	{attribute 'export' := '("archive":"True","name":"АОсс: АОсс от оператора","alarm":("type":"crs","action":"АОсс"),"subsystem":"Внешние источники","condition":("set":"TRUE","reset":"FALSE","active":"btn.AOss.out","fault":"FALSE"))'}
	btn_AOss : Tcrs:= (subsystem_num := 1, type_num := 1); //АОсс: АОсс от оператора//ALG/Внешние источники
	{attribute 'export' := '("archive":"True","name":"АОбс: АОбс от оператора","alarm":("type":"crs","action":"АОбс"),"subsystem":"Внешние источники","condition":("set":"TRUE","reset":"FALSE","active":"btn.AObs.out","fault":"FALSE"))'}
	btn_AObs : Tcrs:= (subsystem_num := 1, type_num := 2); //АОбс: АОбс от оператора//ALG/Внешние источники
	{attribute 'export' := '("archive":"True","name":"АОсс: АОсс по технологическим условиям","alarm":("type":"crs","action":"АОсс"),"subsystem":"Внешние источники","condition":("set":"TRUE","reset":"FALSE","active":"alg.AOss_tech","fault":"FALSE"))'}
	AOss_tech : Tcrs:= (subsystem_num := 1, type_num := 1); //АОсс: АОсс по технологическим условиям//ALG/Внешние источники
	{attribute 'export' := '("archive":"True","name":"АОбс: АОбс по технологическим условиям","alarm":("type":"crs","action":"АОбс"),"subsystem":"Внешние источники","condition":("set":"TRUE","reset":"FALSE","active":"alg.AOss_tech","fault":"FALSE"))'}
	AObs_tech : Tcrs:= (subsystem_num := 1, type_num := 2); //АОбс: АОбс по технологическим условиям//ALG/Внешние источники
	{attribute 'export' := '("archive":"True","name":"АОсс: Кнопка АО на ПРУ","alarm":("type":"crs","action":"АОсс"),"subsystem":"Внешние источники","condition":("set":"TRUE","reset":"FALSE","active":"dipar.AO_PRU_1.value OR dipar.AO_PRU_2.value","fault":"dipar.AO_PRU_1.flt OR dipar.AO_PRU_2.flt"))'}
	AO_PRU : Tcrs:= (subsystem_num := 1, type_num := 1); //АОсс: Кнопка АО на ПРУ//ALG/Внешние источники
	{attribute 'export' := '("archive":"True","name":"АОсс: АО от кнопки \"АО\" блока автоматики ГПА","alarm":("type":"crs","action":"АОсс"),"subsystem":"Внешние источники","condition":("set":"TRUE","reset":"FALSE","active":"dipar.AO_BA.value","fault":"dipar.AO_BA.flt"))'}
	AO_BA : Tcrs:= (subsystem_num := 1, type_num := 1); //АОсс: АО от кнопки "АО" блока автоматики ГПА//DI/Внешние источники
	{attribute 'export' := '("archive":"True","name":"АОсс: БЭАО сработал","alarm":("type":"crs","action":"АОсс"),"subsystem":"Внешние источники","condition":("set":"TRUE","reset":"FALSE","active":"dipar.BEAO.value","fault":"dipar.BEAO.flt"))'}
	BEAO : Tcrs:= (subsystem_num := 1, type_num := 1); //АОсс: БЭАО сработал//DI/Внешние источники
	{attribute 'export' := '("archive":"True","name":"АОбс: Самопроизвольное закрытие СК","alarm":("type":"crs","action":"АОбс"),"subsystem":"Блок двигателя","condition":("set":"FuelReg.fReg.isFire","reset":"NOT am.SK.on","active":"NOT dipar.SK_ON.value","fault":"dipar.SK_ON.flt"))'}
	Causeless_SK : Tcrs:= (subsystem_num := 2, type_num := 2); //АОбс: Самопроизвольное закрытие СК//ALG/Блок двигателя
	{attribute 'export' := '("archive":"True","name":"АОсс: Помпаж двигателя","alarm":("type":"crs","action":"АОсс"),"subsystem":"Блок двигателя","condition":("set":"TRUE","reset":"FALSE","active":"dipar.SurgeD.value","fault":"dipar.SurgeD.flt"))'}
	SurgeD : Tcrs:= (subsystem_num := 2, type_num := 1); //АОсс: Помпаж двигателя//DI/Блок двигателя
	{attribute 'export' := '("archive":"True","name":"АОсс: Опасная вибрация двигателя","alarm":("type":"crs","action":"АОсс"),"subsystem":"Блок двигателя","condition":("set":"TRUE","reset":"FALSE","active":"dipar.Vs_D_Av.value","fault":"dipar.Vs_D_Av.flt"))'}
	Vs_D_Av : Tcrs:= (subsystem_num := 2, type_num := 1); //АОсс: Опасная вибрация двигателя//DI/Блок двигателя
	{attribute 'export' := '("archive":"True","name":"АОбс: Авар.-выс. Вибрация ТК","alarm":("type":"crs","action":"АОбс"),"subsystem":"Блок двигателя","condition":("set":"TRUE","reset":"FALSE","active":"aipar.Vstk.setpoint.HH","fault":"aipar.Vstk.flt"))'}
	Vstk_HH : Tcrs:= (subsystem_num := 2, type_num := 2); //АОбс: Авар.-выс. Вибрация ТК//> 60/Блок двигателя
	{attribute 'export' := '("archive":"True","name":"АОсс: Авар.-выс. Вибрация СТ","alarm":("type":"crs","action":"АОсс"),"subsystem":"Блок двигателя","condition":("set":"TRUE","reset":"FALSE","active":"aipar.Vsst.setpoint.HH","fault":"aipar.Vsst.flt"))'}
	Vsst_HH : Tcrs:= (subsystem_num := 2, type_num := 1); //АОсс: Авар.-выс. Вибрация СТ//> 60/Блок двигателя
	{attribute 'export' := '("archive":"True","name":"АОбс: КПВ234 не закрыты","alarm":("type":"crs","action":"АОбс"),"subsystem":"Блок двигателя","condition":("set":"alg.KPV234_wOpen","reset":"NOT alg.KPV234_wOpen","active":"NOT ( dipar.KPV2_off.value AND dipar.KPV3_off.value AND dipar.KPV4_off.value )","fault":"dipar.KPV2_off.flt OR dipar.KPV3_off.flt OR dipar.KPV4_off.flt"))'}
	KPV234_wOpen : Tcrs:= (subsystem_num := 2, type_num := 2, pt := t#1s0ms); //АОбс: КПВ234 не закрыты//ALG/Блок двигателя
	{attribute 'export' := '("archive":"True","name":"АОбс: КПВ15 не закрыты","alarm":("type":"crs","action":"АОбс"),"subsystem":"Блок двигателя","condition":("set":"alg.KPV15_wOpen","reset":"NOT alg.KPV15_wOpen","active":"NOT ( dipar.KPV1_off.value AND dipar.KPV5_off.value )","fault":"dipar.KPV1_off.flt OR dipar.KPV5_off.flt"))'}
	KPV15_wOpen : Tcrs:= (subsystem_num := 2, type_num := 2, pt := t#1s0ms); //АОбс: КПВ15 не закрыты//ALG/Блок двигателя
	{attribute 'export' := '("archive":"True","name":"АОбс: КПВ15 не открыты","alarm":("type":"crs","action":"АОбс"),"subsystem":"Блок двигателя","condition":("set":"alg.KPV15_nOpen","reset":"NOT alg.KPV15_nOpen","active":"NOT ( dipar.KPV1_ON.value AND dipar.KPV5_ON.value )","fault":"dipar.KPV1_ON.flt OR dipar.KPV5_ON.flt"))'}
	KPV15_nOpen : Tcrs:= (subsystem_num := 2, type_num := 2, pt := t#1s0ms); //АОбс: КПВ15 не открыты//ALG/Блок двигателя
	{attribute 'export' := '("archive":"True","name":"АОсс: Авар.-выс. Обороты СТ > 9300 об/мин","alarm":("type":"crs","action":"АОсс"),"subsystem":"Блок двигателя","condition":("set":"TRUE","reset":"FALSE","active":"acpar.Nst.setpoint.HH","fault":"FALSE"))'}
	Nst_HH : Tcrs:= (subsystem_num := 2, type_num := 1); //АОсс: Авар.-выс. Обороты СТ > 9300 об/мин//> 9000 об/мин/Блок двигателя
	{attribute 'export' := '("archive":"True","name":"АОбс: Авар.-выс. Обороты ТК > 8400 об/мин","alarm":("type":"crs","action":"АОбс"),"subsystem":"Блок двигателя","condition":("set":"TRUE","reset":"FALSE","active":"acpar.Ntk.setpoint.HH","fault":"FALSE"))'}
	Ntk_Av_HH : Tcrs:= (subsystem_num := 2, type_num := 2); //АОбс: Авар.-выс. Обороты ТК > 8400 об/мин//> 8400 об/мин/Блок двигателя
	{attribute 'export' := '("archive":"True","name":"АОбс: Отказ всех датчиков ЧВ ТК","alarm":("type":"crs","action":"АОбс"),"subsystem":"Блок двигателя","condition":("set":"TRUE","reset":"FALSE","active":"aipar.Ntk_1.flt AND aipar.Ntk_2.flt OR acpar.Ntk.flt","fault":"FALSE"))'}
	Ntk_flt : Tcrs:= (subsystem_num := 2, type_num := 2); //АОбс: Отказ всех датчиков ЧВ ТК//ALG/Блок двигателя
	{attribute 'export' := '("archive":"True","name":"АОбс: Отказ всех датчиков ЧВ СТ","alarm":("type":"crs","action":"АОбс"),"subsystem":"Блок двигателя","condition":("set":"TRUE","reset":"FALSE","active":"aipar.Nst_1.flt AND aipar.Nst_2.flt OR acpar.Nst.flt","fault":"FALSE"))'}
	Nst_flt : Tcrs:= (subsystem_num := 2, type_num := 2); //АОбс: Отказ всех датчиков ЧВ СТ//ALG/Блок двигателя
	{attribute 'export' := '("archive":"True","name":"АОбс: Авар.-выс. Температура газа на входе СТ","alarm":("type":"crs","action":"АОбс"),"subsystem":"Блок двигателя","condition":("set":"TRUE","reset":"FALSE","active":"acpar.Tg_inST.setpoint.HH","fault":"FALSE"))'}
	Tg_inST_HH : Tcrs:= (subsystem_num := 2, type_num := 2); //АОбс: Авар.-выс. Температура газа на входе СТ//> 670 °С/Блок двигателя
	{attribute 'export' := '("archive":"True","name":"АОсс: Пожар ОД","alarm":("type":"crs","action":"АОсс"),"subsystem":"Блок двигателя","condition":("set":"TRUE","reset":"FALSE","active":"dipar.Fire_OD.value","fault":"dipar.Fire_OD.flt"))'}
	Fire_OD : Tcrs:= (subsystem_num := 2, type_num := 1); //АОсс: Пожар ОД//DI/Блок двигателя
	{attribute 'export' := '("archive":"True","name":"АОбс: Авар.-выс. Высокая неравномерность 1-ой термопары","alarm":("type":"crs","action":"АОбс"),"subsystem":"Блок двигателя","condition":("set":"am.SK.isON","reset":"am.SK.isOFF","active":"ABS ( acpar.Tg_inST.value - aipar.Tg_inST_1.value ) > 100.0","fault":"aipar.Tg_inST_1.flt"))'}
	Tg1_inSTdistort_HH : Tcrs:= (subsystem_num := 2, type_num := 2); //АОбс: Авар.-выс. Высокая неравномерность 1-ой термопары//<> 100 °С/Блок двигателя
	{attribute 'export' := '("archive":"True","name":"АОбс: Авар.-выс. Высокая неравномерность 2-ой термопары","alarm":("type":"crs","action":"АОбс"),"subsystem":"Блок двигателя","condition":("set":"am.SK.isON","reset":"am.SK.isOFF","active":"ABS ( acpar.Tg_inST.value - aipar.Tg_inST_2.value ) > 100.0","fault":"aipar.Tg_inST_2.flt"))'}
	Tg2_inSTdistort_HH : Tcrs:= (subsystem_num := 2, type_num := 2); //АОбс: Авар.-выс. Высокая неравномерность 2-ой термопары//<> 100 °С/Блок двигателя
	{attribute 'export' := '("archive":"True","name":"АОбс: Авар.-выс. Высокая неравномерность 3-ой термопары","alarm":("type":"crs","action":"АОбс"),"subsystem":"Блок двигателя","condition":("set":"am.SK.isON","reset":"am.SK.isOFF","active":"ABS ( acpar.Tg_inST.value - aipar.Tg_inST_3.value ) > 100.0","fault":"aipar.Tg_inST_3.flt"))'}
	Tg3_inSTdistort_HH : Tcrs:= (subsystem_num := 2, type_num := 2); //АОбс: Авар.-выс. Высокая неравномерность 3-ой термопары//<> 100 °С/Блок двигателя
	{attribute 'export' := '("archive":"True","name":"АОбс: Авар.-выс. Высокая неравномерность 4-ой термопары","alarm":("type":"crs","action":"АОбс"),"subsystem":"Блок двигателя","condition":("set":"am.SK.isON","reset":"am.SK.isOFF","active":"ABS ( acpar.Tg_inST.value - aipar.Tg_inST_4.value ) > 100.0","fault":"aipar.Tg_inST_4.flt"))'}
	Tg4_inSTdistort_HH : Tcrs:= (subsystem_num := 2, type_num := 2); //АОбс: Авар.-выс. Высокая неравномерность 4-ой термопары//<> 100 °С/Блок двигателя
	{attribute 'export' := '("archive":"True","name":"АОбс: Авар.-выс. Высокая неравномерность 5-ой термопары","alarm":("type":"crs","action":"АОбс"),"subsystem":"Блок двигателя","condition":("set":"am.SK.isON","reset":"am.SK.isOFF","active":"ABS ( acpar.Tg_inST.value - aipar.Tg_inST_5.value ) > 100.0","fault":"aipar.Tg_inST_5.flt"))'}
	Tg5_inSTdistort_HH : Tcrs:= (subsystem_num := 2, type_num := 2); //АОбс: Авар.-выс. Высокая неравномерность 5-ой термопары//<> 100 °С/Блок двигателя
	{attribute 'export' := '("archive":"True","name":"АОбс: Авар.-выс. Высокая неравномерность 6-ой термопары","alarm":("type":"crs","action":"АОбс"),"subsystem":"Блок двигателя","condition":("set":"am.SK.isON","reset":"am.SK.isOFF","active":"ABS ( acpar.Tg_inST.value - aipar.Tg_inST_6.value ) > 100.0","fault":"aipar.Tg_inST_6.flt"))'}
	Tg6_inSTdistort_HH : Tcrs:= (subsystem_num := 2, type_num := 2); //АОбс: Авар.-выс. Высокая неравномерность 6-ой термопары//<> 100 °С/Блок двигателя
	{attribute 'export' := '("archive":"True","name":"АОбс: Отказ 4-х и более термопар","alarm":("type":"crs","action":"АОбс"),"subsystem":"Блок двигателя","condition":("set":"TRUE","reset":"FALSE","active":"alg.TstInWork < 3","fault":"FALSE"))'}
	Tg_inSTflt : Tcrs:= (subsystem_num := 2, type_num := 2); //АОбс: Отказ 4-х и более термопар//ALG/Блок двигателя
	{attribute 'export' := '("archive":"True","name":"АОбс: Нет розжига на пуске","alarm":("type":"crs","action":"АОбс"),"subsystem":"Блок двигателя","condition":("set":"alg.sh_nIgnition","reset":"NOT alg.sh_nIgnition","active":"NOT FuelReg.fReg.isFire","fault":"FALSE"))'}
	nIgnition : Tcrs:= (subsystem_num := 2, type_num := 2, pt := t#10s0ms); //АОбс: Нет розжига на пуске//DI/Блок двигателя
	{attribute 'export' := '("archive":"True","name":"АОбс: Погасание факела","alarm":("type":"crs","action":"АОбс"),"subsystem":"Блок двигателя","condition":("set":"TRUE","reset":"FALSE","active":"FuelReg.fReg.noFire","fault":"FALSE"))'}
	Fire_flt : Tcrs:= (subsystem_num := 2, type_num := 2); //АОбс: Погасание факела//ALG/Блок двигателя
	{attribute 'export' := '("archive":"True","name":"АОбс: Отсутствие раскрутки ТК","alarm":("type":"crs","action":"АОбс"),"subsystem":"Блок двигателя","condition":("set":"alg.sh_nBoost","reset":"NOT alg.sh_nBoost","active":"acpar.Ntk.value < 5600","fault":"acpar.Ntk.flt"))'}
	Ntk_nBoost : Tcrs:= (subsystem_num := 2, type_num := 2, pt := t#10s0ms); //АОбс: Отсутствие раскрутки ТК//DI/Блок двигателя
	{attribute 'export' := '("archive":"True","name":"АОбс: Рассогласование ДГ","alarm":("type":"crs","action":"АОбс"),"subsystem":"Блок двигателя","condition":("set":"am.SK.on","reset":"NOT am.SK.on","active":"ABS(aopar.DG_set.value - aipar.DG_Pos.value) >= 1.0","fault":"aipar.DG_Pos.flt"))'}
	DGdistort : Tcrs:= (subsystem_num := 2, type_num := 2, pt := t#2s0ms); //АОбс: Рассогласование ДГ//ALG/Блок двигателя
	{attribute 'export' := '("archive":"True","name":"АОбс: Авар.-выс. Давление воздуха за 14-й ступенью осевого компрессора","alarm":("type":"crs","action":"АОбс"),"subsystem":"Блок двигателя","condition":("set":"TRUE","reset":"FALSE","active":"aipar.Pa_out14.setpoint.HH","fault":"aipar.Pa_out14.flt"))'}
	Pa_out14_HH : Tcrs:= (subsystem_num := 2, type_num := 2); //АОбс: Авар.-выс. Давление воздуха за 14-й ступенью осевого компрессора//> 2.0/Блок двигателя
	{attribute 'export' := '("archive":"True","name":"АОбс: Неисправность БЗА на пуске","alarm":("type":"crs","action":"АОбс"),"subsystem":"Блок двигателя","condition":("set":"( acpar.Ntk.value > BZA.Ntk_SetUp ) AND ( acpar.Nst.value > BZA.Nst_SetUp )","reset":"NOT tch.GTDstart.value","active":"NOT dipar.BZA_ready_1.value OR NOT dipar.BZA_ready_2.value","fault":"FALSE"))'}
	BZA_ready_2 : Tcrs:= (subsystem_num := 2, type_num := 2); //АОбс: Неисправность БЗА на пуске//DI/Блок двигателя
	{attribute 'export' := '("archive":"True","name":"АОсс: БЗА: Авария","alarm":("type":"crs","action":"АОсс"),"subsystem":"Блок двигателя","condition":("set":"TRUE","reset":"FALSE","active":"dipar.BZA_alr.value","fault":"dipar.BZA_alr.flt"))'}
	BZA_alr : Tcrs:= (subsystem_num := 2, type_num := 1); //АОсс: БЗА: Авария//DI/Блок двигателя
	{attribute 'export' := '("archive":"True","name":"АОбс: Давление масла смазки ТК аварийное","alarm":("type":"crs","action":"АОбс"),"subsystem":"Маслосистема двигателя","condition":("set":"alg.sh_PmGTD","reset":"NOT alg.sh_PmGTD","active":"dipar.Pm_TK_An.value","fault":"dipar.Pm_TK_An.flt"))'}
	Pm_TK_An : Tcrs:= (subsystem_num := 3, type_num := 2, pt := t#3s0ms); //АОбс: Давление масла смазки ТК аварийное//DI/Маслосистема двигателя
	{attribute 'export' := '("archive":"True","name":"АОбс: Давление масла смазки СТ аварийное","alarm":("type":"crs","action":"АОбс"),"subsystem":"Маслосистема двигателя","condition":("set":"alg.sh_PmGTD","reset":"NOT alg.sh_PmGTD","active":"dipar.Pm_ST_An.value","fault":"dipar.Pm_ST_An.flt"))'}
	Pm_ST_An : Tcrs:= (subsystem_num := 3, type_num := 2, pt := t#3s0ms); //АОбс: Давление масла смазки СТ аварийное//DI/Маслосистема двигателя
	{attribute 'export' := '("archive":"True","name":"АОбс: Авар.-выс. Температура масла на выходе двигателя","alarm":("type":"crs","action":"АОбс"),"subsystem":"Маслосистема двигателя","condition":("set":"TRUE","reset":"FALSE","active":"aipar.Tm_outD.setpoint.HH","fault":"aipar.Tm_outD.flt"))'}
	Tm_outD_HH : Tcrs:= (subsystem_num := 3, type_num := 2, pt := t#1s0ms); //АОбс: Авар.-выс. Температура масла на выходе двигателя//> 85 °С/Маслосистема двигателя
	{attribute 'export' := '("archive":"True","name":"АОсс: Стружка в масле на выходе Д","alarm":("type":"crs","action":"АОсс"),"subsystem":"Маслосистема двигателя","condition":("set":"TRUE","reset":"FALSE","active":"dipar.Chip_outD.value","fault":"dipar.Chip_outD.flt"))'}
	Chip_outD : Tcrs:= (subsystem_num := 3, type_num := 1); //АОсс: Стружка в масле на выходе Д//DI/Маслосистема двигателя
	{attribute 'export' := '("archive":"True","name":"АОбс: Аварийное давление газа до крана 13","alarm":("type":"crs","action":"АОбс"),"subsystem":"Воздушный стартер","condition":("set":"alg.sh_Pg_InKR13","reset":"NOT alg.sh_Pg_InKR13","active":"dipar.Pg_InKR13.value","fault":"dipar.Pg_InKR13.flt"))'}
	Pg_InKR13 : Tcrs:= (subsystem_num := 4, type_num := 2, pt := t#10s0ms); //АОбс: Аварийное давление газа до крана 13//DI/Воздушный стартер
	{attribute 'export' := '("archive":"True","name":"АОбс: Давление масла смазки воздушного стартера высокий уровень","alarm":("type":"crs","action":"АОбс"),"subsystem":"Воздушный стартер","condition":("set":"TRUE","reset":"FALSE","active":"dipar.Pm_Starter_Av.value","fault":"dipar.Pm_Starter_Av.flt"))'}
	Pm_Starter_Av : Tcrs:= (subsystem_num := 4, type_num := 2, pt := t#10s0ms); //АОбс: Давление масла смазки воздушного стартера высокий уровень//DI/Воздушный стартер
	{attribute 'export' := '("archive":"True","name":"АОбс: Давление масла смазки воздушного стартера низкий уровень","alarm":("type":"crs","action":"АОбс"),"subsystem":"Воздушный стартер","condition":("set":"alg.sh_Starter","reset":"am.KR13.isOFF","active":"dipar.Pm_Starter_An.value","fault":"dipar.Pm_Starter_An.flt"))'}
	Pm_Starter_An : Tcrs:= (subsystem_num := 4, type_num := 2); //АОбс: Давление масла смазки воздушного стартера низкий уровень//DI/Воздушный стартер
	{attribute 'export' := '("archive":"True","name":"АОбс: Давление газа перед дозатором газа Аварийное","alarm":("type":"crs","action":"АОбс"),"subsystem":"Блок топливного газа","condition":("set":"alg.sh_TG","reset":"NOT alg.sh_TG","active":"dipar.Ptg_inDG_An.value","fault":"dipar.Ptg_inDG_An.flt"))'}
	Ptg_inDG_An : Tcrs:= (subsystem_num := 6, type_num := 2, pt := t#1s0ms); //АОбс: Давление газа перед дозатором газа Аварийное//DI/Блок топливного газа
	{attribute 'export' := '("archive":"True","name":"АОсс: dP перед форсунками камеры сгорания >10кПа","alarm":("type":"crs","action":"АОсс"),"subsystem":"Блок топливного газа","condition":("set":"am.SK.isOFF AND ( acpar.Ntk.value < 100 )","reset":"am.SK.isON","active":"dipar.dP_F_Pv.value","fault":"dipar.dP_F_Pv.flt"))'}
	dP_F_Pv : Tcrs:= (subsystem_num := 6, type_num := 1, pt := t#3s0ms); //АОсс: dP перед форсунками камеры сгорания >10кПа//DI/Блок топливного газа
	{attribute 'export' := '("archive":"True","name":"АОбс: Аварийное давление масла перед ДГ","alarm":("type":"crs","action":"АОбс"),"subsystem":"Блок топливного газа","condition":("set":"alg.sh_SAR","reset":"NOT alg.sh_SAR","active":"dipar.Pm_SAR_An.value","fault":"dipar.Pm_SAR_An.flt"))'}
	Pm_SAR_An : Tcrs:= (subsystem_num := 6, type_num := 2, pt := t#1s0ms); //АОбс: Аварийное давление масла перед ДГ//DI/Блок топливного газа
	{attribute 'export' := '("archive":"True","name":"АОбс: Авар.-низ. Давление топливного газа перед ТРК","alarm":("type":"crs","action":"АОбс"),"subsystem":"Блок топливного газа","condition":("set":"alg.sh_TG","reset":"NOT alg.sh_TG","active":"aipar.Ptg_inTRK.setpoint.LL","fault":"aipar.Ptg_inTRK.flt"))'}
	Ptg_inTRK_LL : Tcrs:= (subsystem_num := 6, type_num := 2, pt := t#3s0ms); //АОбс: Авар.-низ. Давление топливного газа перед ТРК//< 10 кгс/см2/Блок топливного газа
	{attribute 'export' := '("archive":"True","name":"АОсс: Помпаж нагнетателя","alarm":("type":"crs","action":"АОсс"),"subsystem":"Компрессорная установка/блок нагнетателя","condition":("set":"TRUE","reset":"FALSE","active":"s_tunpar.ASprot.surge","fault":"s_tunpar.ASprot.surgeAlertBrk"))'}
	AS_Av : Tcrs:= (subsystem_num := 9, type_num := 1); //АОсс: Помпаж нагнетателя//DI/Компрессорная установка/блок нагнетателя
	{attribute 'export' := '("archive":"True","name":"АОсс: Авар.-низ. Перепад давления “масло-газ”","alarm":("type":"crs","action":"АОсс"),"subsystem":"Компрессорная установка/блок нагнетателя","condition":("set":"alg.sh_dPmg","reset":"NOT alg.sh_dPmg","active":"aipar.dPmg.setpoint.LL OR dipar.dPmg_An.value","fault":"dipar.dPmg_An.flt OR aipar.dPmg.flt OR NOT aipar.dPmg.setpoint.isLL"))'}
	dPmg_LL : Tcrs:= (subsystem_num := 9, type_num := 1); //АОсс: Авар.-низ. Перепад давления “масло-газ”//< 0.3 кгс/см2/Компрессорная установка/блок нагнетателя
	{attribute 'export' := '("archive":"True","name":"АОсс: Давление масла смазки Н аварийное","alarm":("type":"crs","action":"АОсс"),"subsystem":"Компрессорная установка/блок нагнетателя","condition":("set":"alg.sh_PmN","reset":"NOT alg.sh_PmN","active":"dipar.Pm_N_An.value","fault":"dipar.Pm_N_An.flt"))'}
	Pm_N_An : Tcrs:= (subsystem_num := 9, type_num := 1, pt := t#3s0ms); //АОсс: Давление масла смазки Н аварийное//DI/Компрессорная установка/блок нагнетателя
	{attribute 'export' := '("archive":"True","name":"АОсс: Аварийный осевой сдвиг ротора Н","alarm":("type":"crs","action":"АОсс"),"subsystem":"Компрессорная установка/блок нагнетателя","condition":("set":"TRUE","reset":"FALSE","active":"dipar.Zs_Nl.value","fault":"dipar.Zs_Nl.flt"))'}
	Zs_Nl : Tcrs:= (subsystem_num := 9, type_num := 1); //АОсс: Аварийный осевой сдвиг ротора Н//DI/Компрессорная установка/блок нагнетателя
	{attribute 'export' := '("archive":"True","name":"АОбс: Кран 6 закрыт на пуске","alarm":("type":"crs","action":"АОбс"),"subsystem":"Компрессорная установка/блок нагнетателя","condition":("set":"acpar.Nst.value > 300.0  AND Start_D.drm.active","reset":"acpar.Nst.value < 300.0 OR NOT Start_D.drm.active","active":"dipar.Kr6_off.value","fault":"dipar.Kr6_off.flt"))'}
	Kr6_off_start : Tcrs:= (subsystem_num := 9, type_num := 2, pt := t#3s0ms); //АОбс: Кран 6 закрыт на пуске//ALG/Компрессорная установка/блок нагнетателя
	{attribute 'export' := '("archive":"True","name":"АОбс: Самопроизвольное закрытие крана 1","alarm":("type":"crs","action":"АОбс"),"subsystem":"Газовая обвязка","condition":("set":"alg.work","reset":"NOT alg.work","active":"NOT dipar.Kr1_ON.value","fault":"FALSE"))'}
	Causeless_KR1_off : Tcrs:= (subsystem_num := 11, type_num := 2, pt := t#3s0ms); //АОбс: Самопроизвольное закрытие крана 1//ALG/Газовая обвязка
	{attribute 'export' := '("archive":"True","name":"АОбс: Самопроизвольное закрытие крана 2","alarm":("type":"crs","action":"АОбс"),"subsystem":"Газовая обвязка","condition":("set":"alg.work","reset":"NOT alg.work","active":"NOT dipar.Kr2_ON.value AND dipar.Kr6_off.value","fault":"FALSE"))'}
	Causeless_KR2_off : Tcrs:= (subsystem_num := 11, type_num := 2, pt := t#3s0ms); //АОбс: Самопроизвольное закрытие крана 2//ALG/Газовая обвязка
	{attribute 'export' := '("archive":"True","name":"АОбс: Самопроизвольное закрытие крана 6","alarm":("type":"crs","action":"АОбс"),"subsystem":"Газовая обвязка","condition":("set":"alg.work","reset":"NOT alg.work","active":"NOT dipar.Kr6_ON.value AND (NOT dipar.Kr2_ON.value OR dipar.Kr2_off.value)","fault":"FALSE"))'}
	Causeless_KR6_off : Tcrs:= (subsystem_num := 11, type_num := 2, pt := t#3s0ms); //АОбс: Самопроизвольное закрытие крана 6//ALG/Газовая обвязка
	{attribute 'export' := '("archive":"True","name":"АОбс: Самопроизвольная перестановка кранов 10, 11","alarm":("type":"crs","action":"АОбс"),"subsystem":"Газовая обвязка","condition":("set":"am.KR15.on","reset":"NOT am.KR15.on","active":"NOT ( dipar.Kr10_off.value AND dipar.Kr11_ON.value )","fault":"FALSE"))'}
	Causeless_KR10_11 : Tcrs:= (subsystem_num := 11, type_num := 2, pt := t#1s0ms); //АОбс: Самопроизвольная перестановка кранов 10, 11//ALG/Газовая обвязка
END_VAR
(* global variable list ppu *)
{region INFO}
(*
 Назначение: Признаки срабатывания предпусковых условий
 Автор:  /Andrey/ 24.06.2025 16:50:31
 Версия: v00.00.22
 Проект: KA107__GPA2
*)
{endregion}
{attribute 'qualified_only'}
{attribute 'symbol' := 'read'}
VAR_GLOBAL
	{attribute 'symbol' := 'none'}
	common: Talarm; //Общий сигнал для VAR_STAT
	{attribute 'export' := '("archive":"True","name":"Контроль ХР")'}
	check_HR: Ttch; //Контроль ХР
	{attribute 'export' := '("archive":"True","name":"Контроль ГР")'}
	check_GR: Ttch; //Контроль ГР
	{attribute 'symbol' := 'none'}
	HR: BOOL; //Условия ХР собраны
	{attribute 'symbol' := 'none'}
	GR: BOOL; //Условия ГР собраны

	{attribute 'export' := '("archive":"True","name":"Есть недеблокированные АС","alarm":("type":"ppu","action":"ХР"),"condition":("set":"TRUE","reset":"FALSE","active":"crs.common.aggregated"))'}
	crs_aggregated : Talarm:= (subsystem_num := 1, type_num := 4); //Есть недеблокированные АС//Внутренний сигнал/Внешние источники
	{attribute 'export' := '("archive":"True","name":"Расчетная N ротора ГГ > 100 об/мин","alarm":("type":"ppu","action":"ХР"),"condition":("set":"TRUE","reset":"FALSE","active":"acpar.Ntk.value > 100.0"))'}
	evNvd_H : Talarm:= (subsystem_num := 2, type_num := 4); //Расчетная N ротора ГГ > 100 об/мин//> 100 об/мин/Блок двигателя
	{attribute 'export' := '("archive":"True","name":"Расчетная N ротора СТ > 100 об/мин","alarm":("type":"ppu","action":"ХР"),"condition":("set":"TRUE","reset":"FALSE","active":"acpar.Nst.value > 100.0"))'}
	evNst_H : Talarm:= (subsystem_num := 2, type_num := 4); //Расчетная N ротора СТ > 100 об/мин//> 100 об/мин/Блок двигателя
	{attribute 'export' := '("archive":"True","name":"Нет сигнала: СК закрыт","alarm":("type":"ppu","action":"ХР"),"condition":("set":"TRUE","reset":"FALSE","active":"NOT dipar.SK_off.value"))'}
	N_SK_off : Talarm:= (subsystem_num := 2, type_num := 4); //Нет сигнала: СК закрыт//Нет DI/Блок двигателя
	{attribute 'export' := '("archive":"True","name":"Загазованность контейнеров выше нормы","alarm":("type":"ppu","action":"ХР"),"condition":("set":"TRUE","reset":"FALSE","active":"dipar.Zagaz_OD_Pv.value"))'}
	Zagaz_OD_Pv : Talarm:= (subsystem_num := 2, type_num := 4); //Загазованность контейнеров выше нормы//DI/Блок двигателя
	{attribute 'export' := '("archive":"True","name":"Сигнализатор обледенения","alarm":("type":"ppu","action":"ГР"),"condition":("set":"TRUE","reset":"FALSE","active":"dipar.Ace_alr.value"))'}
	Ace_alr : Talarm:= (subsystem_num := 2, type_num := 4); //Сигнализатор обледенения//DI/Блок двигателя
	{attribute 'export' := '("archive":"True","name":"Нет сигнала: ТРК: готовность","alarm":("type":"ppu","action":"ХР"),"condition":("set":"TRUE","reset":"FALSE","active":"NOT dipar.TRKready.value"))'}
	N_TRKready : Talarm:= (subsystem_num := 2, type_num := 4); //Нет сигнала: ТРК: готовность//Нет DI/Блок двигателя
	{attribute 'export' := '("archive":"True","name":"ТРК: авария","alarm":("type":"ppu","action":"ХР"),"condition":("set":"TRUE","reset":"FALSE","active":"dipar.TRKalr.value"))'}
	TRKalr : Talarm:= (subsystem_num := 2, type_num := 4); //ТРК: авария//DI/Блок двигателя
	{attribute 'export' := '("archive":"True","name":"Нет сигнала: БЗА: Готовность 1","alarm":("type":"ppu","action":"ГР"),"condition":("set":"TRUE","reset":"FALSE","active":"NOT dipar.BZA_ready_1.value"))'}
	N_BZA_ready_1 : Talarm:= (subsystem_num := 2, type_num := 4); //Нет сигнала: БЗА: Готовность 1//Нет DI/Блок двигателя
	{attribute 'export' := '("archive":"True","name":"Неисправность БЗА","alarm":("type":"ppu","action":"ГР"),"condition":("set":"TRUE","reset":"FALSE","active":"dipar.BZA_ready_1.value AND dipar.BZA_ready_2.value"))'}
	BZA_flt : Talarm:= (subsystem_num := 2, type_num := 4); //Неисправность БЗА//ALG/Блок двигателя
	{attribute 'export' := '("archive":"True","name":"Пониж. Температура масла в баке Д и Н","alarm":("type":"ppu","action":"ХР"),"condition":("set":"TRUE","reset":"FALSE","active":"aipar.Tm_MB.setpoint.L"))'}
	Tm_MB_L : Talarm:= (subsystem_num := 3, type_num := 4); //Пониж. Температура масла в баке Д и Н//< 5 °С/Маслосистема двигателя
	{attribute 'export' := '("archive":"True","name":"Кран №9 не открыт","alarm":("type":"ppu","action":"ХР"),"condition":("set":"TRUE","reset":"FALSE","active":"NOT dipar.Kr9_ON.value OR dipar.Kr9_off.value"))'}
	Kr9_ON : Talarm:= (subsystem_num := 6, type_num := 4); //Кран №9 не открыт//ALG/Блок топливного газа
	{attribute 'export' := '("archive":"True","name":"Кран №12 не закрыт","alarm":("type":"ppu","action":"ХР"),"condition":("set":"TRUE","reset":"FALSE","active":"NOT dipar.Kr12_off.value OR dipar.Kr12_ON.value"))'}
	Kr12_off : Talarm:= (subsystem_num := 6, type_num := 4); //Кран №12 не закрыт//ALG/Блок топливного газа
	{attribute 'export' := '("archive":"True","name":"Кран №10 не открыт","alarm":("type":"ppu","action":"ХР"),"condition":("set":"TRUE","reset":"FALSE","active":"NOT dipar.Kr10_ON.value OR dipar.Kr10_off.value"))'}
	Kr10_ON : Talarm:= (subsystem_num := 7, type_num := 4); //Кран №10 не открыт//ALG/Блок пускового газа
	{attribute 'export' := '("archive":"True","name":"Кран №11 не закрыт","alarm":("type":"ppu","action":"ХР"),"condition":("set":"TRUE","reset":"FALSE","active":"NOT dipar.Kr11_off.value OR dipar.Kr11_ON.value"))'}
	Kr11_off : Talarm:= (subsystem_num := 7, type_num := 4); //Кран №11 не закрыт//ALG/Блок пускового газа
	{attribute 'export' := '("archive":"True","name":"Пониж. Температура масла в баке уплотнения","alarm":("type":"ppu","action":"ХР"),"condition":("set":"TRUE","reset":"FALSE","active":"aipar.Tm_MBU.setpoint.L"))'}
	Tm_MBU_L : Talarm:= (subsystem_num := 9, type_num := 4); //Пониж. Температура масла в баке уплотнения//< 5 °С/Компрессорная установка/блок нагнетателя
	{attribute 'export' := '("archive":"True","name":"Нет сигнала: Предохранитель UCP1-XTFU1:1 питания модулей AO исправен","alarm":("type":"ppu","action":"ХР"),"condition":("set":"TRUE","reset":"FALSE","active":"NOT dipar.Fuse_AO_UCP1.value"))'}
	N_Fuse_AO_UCP1 : Talarm:= (subsystem_num := 10, type_num := 4); //Нет сигнала: Предохранитель UCP1-XTFU1:1 питания модулей AO исправен//Нет DI/Блок управления
	{attribute 'export' := '("archive":"True","name":"Нет сигнала: Предохранитель UCP1-XTFU1:2 питания модулей DO исправен","alarm":("type":"ppu","action":"ХР"),"condition":("set":"TRUE","reset":"FALSE","active":"NOT dipar.Fuse_DO_UCP1.value"))'}
	N_Fuse_DO_UCP1 : Talarm:= (subsystem_num := 10, type_num := 4); //Нет сигнала: Предохранитель UCP1-XTFU1:2 питания модулей DO исправен//Нет DI/Блок управления
	{attribute 'export' := '("archive":"True","name":"Нет сигнала: Предохранитель UCP1--XTFU6:1 питания датчиков температуры и влажности","alarm":("type":"ppu","action":"ХР"),"condition":("set":"TRUE","reset":"FALSE","active":"NOT dipar.Fuse_Air_UCP1.value"))'}
	N_Fuse_Air_UCP1 : Talarm:= (subsystem_num := 10, type_num := 4); //Нет сигнала: Предохранитель UCP1--XTFU6:1 питания датчиков температуры и влажности//Нет DI/Блок управления
	{attribute 'export' := '("archive":"True","name":"Нет сигнала: Предохранитель UE1-XTFU1:2 питания модулей DO исправен","alarm":("type":"ppu","action":"ХР"),"condition":("set":"TRUE","reset":"FALSE","active":"NOT dipar.Fuse_DO_UE1.value"))'}
	N_Fuse_DO_UE1 : Talarm:= (subsystem_num := 10, type_num := 4); //Нет сигнала: Предохранитель UE1-XTFU1:2 питания модулей DO исправен//Нет DI/Блок управления
	{attribute 'export' := '("archive":"True","name":"Перегрузка фильтра EV1 (Осн.)","alarm":("type":"ppu","action":"ХР"),"condition":("set":"TRUE","reset":"FALSE","active":"dipar.EV1.value"))'}
	EV1 : Talarm:= (subsystem_num := 10, type_num := 4); //Перегрузка фильтра EV1 (Осн.)//DI/Блок управления
	{attribute 'export' := '("archive":"True","name":"Перегрузка фильтра EV2 (Рез.)","alarm":("type":"ppu","action":"ХР"),"condition":("set":"TRUE","reset":"FALSE","active":"dipar.EV2.value"))'}
	EV2 : Talarm:= (subsystem_num := 10, type_num := 4); //Перегрузка фильтра EV2 (Рез.)//DI/Блок управления
	{attribute 'export' := '("archive":"True","name":"Нет сигнала: Контроль основного ввода питания (-KV1)","alarm":("type":"ppu","action":"ХР"),"condition":("set":"TRUE","reset":"FALSE","active":"NOT dipar.U_main.value"))'}
	N_U_main : Talarm:= (subsystem_num := 10, type_num := 4); //Нет сигнала: Контроль основного ввода питания (-KV1)//Нет DI/Блок управления
	{attribute 'export' := '("archive":"True","name":"Нет сигнала: Контроль резервного ввода питания (-KV2)","alarm":("type":"ppu","action":"ХР"),"condition":("set":"TRUE","reset":"FALSE","active":"NOT dipar.U_res.value"))'}
	N_U_res : Talarm:= (subsystem_num := 10, type_num := 4); //Нет сигнала: Контроль резервного ввода питания (-KV2)//Нет DI/Блок управления
	{attribute 'export' := '("archive":"True","name":"Нет сигнала: Контроль -AG1","alarm":("type":"ppu","action":"ХР"),"condition":("set":"TRUE","reset":"FALSE","active":"NOT dipar.AG1.value"))'}
	N_AG1 : Talarm:= (subsystem_num := 10, type_num := 4); //Нет сигнала: Контроль -AG1//Нет DI/Блок управления
	{attribute 'export' := '("archive":"True","name":"Нет сигнала: Контроль -AG2","alarm":("type":"ppu","action":"ХР"),"condition":("set":"TRUE","reset":"FALSE","active":"NOT dipar.AG2.value"))'}
	N_AG2 : Talarm:= (subsystem_num := 10, type_num := 4); //Нет сигнала: Контроль -AG2//Нет DI/Блок управления
	{attribute 'export' := '("archive":"True","name":"Нет сигнала: Контроль -AG3","alarm":("type":"ppu","action":"ХР"),"condition":("set":"TRUE","reset":"FALSE","active":"NOT dipar.AG3.value"))'}
	N_AG3 : Talarm:= (subsystem_num := 10, type_num := 4); //Нет сигнала: Контроль -AG3//Нет DI/Блок управления
	{attribute 'export' := '("archive":"True","name":"Нет сигнала: Контроль -AG4","alarm":("type":"ppu","action":"ХР"),"condition":("set":"TRUE","reset":"FALSE","active":"NOT dipar.AG4.value"))'}
	N_AG4 : Talarm:= (subsystem_num := 10, type_num := 4); //Нет сигнала: Контроль -AG4//Нет DI/Блок управления
	{attribute 'export' := '("archive":"True","name":"Нет сигнала: Контроль -AG9","alarm":("type":"ppu","action":"ХР"),"condition":("set":"TRUE","reset":"FALSE","active":"NOT dipar.AG9.value"))'}
	N_AG9 : Talarm:= (subsystem_num := 10, type_num := 4); //Нет сигнала: Контроль -AG9//Нет DI/Блок управления
	{attribute 'export' := '("archive":"True","name":"Нет сигнала: Контроль -AG10","alarm":("type":"ppu","action":"ХР"),"condition":("set":"TRUE","reset":"FALSE","active":"NOT dipar.AG10.value"))'}
	N_AG10 : Talarm:= (subsystem_num := 10, type_num := 4); //Нет сигнала: Контроль -AG10//Нет DI/Блок управления
	{attribute 'export' := '("archive":"True","name":"Нет сигнала: Контроль -AG15","alarm":("type":"ppu","action":"ХР"),"condition":("set":"TRUE","reset":"FALSE","active":"NOT dipar.AG15.value"))'}
	N_AG15 : Talarm:= (subsystem_num := 10, type_num := 4); //Нет сигнала: Контроль -AG15//Нет DI/Блок управления
	{attribute 'export' := '("archive":"True","name":"Нет сигнала: Контроль -AG16","alarm":("type":"ppu","action":"ХР"),"condition":("set":"TRUE","reset":"FALSE","active":"NOT dipar.AG16.value"))'}
	N_AG16 : Talarm:= (subsystem_num := 10, type_num := 4); //Нет сигнала: Контроль -AG16//Нет DI/Блок управления
	{attribute 'export' := '("archive":"True","name":"Нет сигнала: Контроль -AG5","alarm":("type":"ppu","action":"ХР"),"condition":("set":"TRUE","reset":"FALSE","active":"NOT dipar.AG5.value"))'}
	N_AG5 : Talarm:= (subsystem_num := 10, type_num := 4); //Нет сигнала: Контроль -AG5//Нет DI/Блок управления
	{attribute 'export' := '("archive":"True","name":"Нет сигнала: Контроль -AG6","alarm":("type":"ppu","action":"ХР"),"condition":("set":"TRUE","reset":"FALSE","active":"NOT dipar.AG6.value"))'}
	N_AG6 : Talarm:= (subsystem_num := 10, type_num := 4); //Нет сигнала: Контроль -AG6//Нет DI/Блок управления
	{attribute 'export' := '("archive":"True","name":"Нет сигнала: Контроль -AG8","alarm":("type":"ppu","action":"ХР"),"condition":("set":"TRUE","reset":"FALSE","active":"NOT dipar.AG8.value"))'}
	N_AG8 : Talarm:= (subsystem_num := 10, type_num := 4); //Нет сигнала: Контроль -AG8//Нет DI/Блок управления
	{attribute 'export' := '("archive":"True","name":"Нет сигнала: Контроль -AG17","alarm":("type":"ppu","action":"ХР"),"condition":("set":"TRUE","reset":"FALSE","active":"NOT dipar.AG17.value"))'}
	N_AG17 : Talarm:= (subsystem_num := 10, type_num := 4); //Нет сигнала: Контроль -AG17//Нет DI/Блок управления
	{attribute 'export' := '("archive":"True","name":"Нет сигнала: Контроль -AG18","alarm":("type":"ppu","action":"ХР"),"condition":("set":"TRUE","reset":"FALSE","active":"NOT dipar.AG18.value"))'}
	N_AG18 : Talarm:= (subsystem_num := 10, type_num := 4); //Нет сигнала: Контроль -AG18//Нет DI/Блок управления
	{attribute 'export' := '("archive":"True","name":"Нет сигнала: Контроль питания ПРУ","alarm":("type":"ppu","action":"ХР"),"condition":("set":"TRUE","reset":"FALSE","active":"NOT dipar.U_PRU.value"))'}
	N_U_PRU : Talarm:= (subsystem_num := 10, type_num := 4); //Нет сигнала: Контроль питания ПРУ//Нет DI/Блок управления
	{attribute 'export' := '("archive":"True","name":"Нет сигнала: Контроль питания ТРК осн.","alarm":("type":"ppu","action":"ХР"),"condition":("set":"TRUE","reset":"FALSE","active":"NOT dipar.Utrk_main.value"))'}
	N_Utrk_main : Talarm:= (subsystem_num := 10, type_num := 4); //Нет сигнала: Контроль питания ТРК осн.//Нет DI/Блок управления
	{attribute 'export' := '("archive":"True","name":"Контроль замыкания на землю питания ИМ","alarm":("type":"ppu","action":"ХР"),"condition":("set":"TRUE","reset":"FALSE","active":"dipar.U_G_AM.value"))'}
	U_G_AM : Talarm:= (subsystem_num := 10, type_num := 4); //Контроль замыкания на землю питания ИМ//DI/Блок управления
	{attribute 'export' := '("archive":"True","name":"Нет сигнала: Контроль питания AI","alarm":("type":"ppu","action":"ХР"),"condition":("set":"TRUE","reset":"FALSE","active":"NOT dipar.U_AI.value"))'}
	N_U_AI : Talarm:= (subsystem_num := 10, type_num := 4); //Нет сигнала: Контроль питания AI//Нет DI/Блок управления
	{attribute 'export' := '("archive":"True","name":"Нет сигнала: Контроль питания DI","alarm":("type":"ppu","action":"ХР"),"condition":("set":"TRUE","reset":"FALSE","active":"NOT dipar.U_DI.value"))'}
	N_U_DI : Talarm:= (subsystem_num := 10, type_num := 4); //Нет сигнала: Контроль питания DI//Нет DI/Блок управления
	{attribute 'export' := '("archive":"True","name":"Нет сигнала: Контроль питания БИЗ","alarm":("type":"ppu","action":"ХР"),"condition":("set":"TRUE","reset":"FALSE","active":"NOT dipar.U_BIZ.value"))'}
	N_U_BIZ : Talarm:= (subsystem_num := 10, type_num := 4); //Нет сигнала: Контроль питания БИЗ//Нет DI/Блок управления
	{attribute 'export' := '("archive":"True","name":"Нет сигнала: Контроль питания ИМ","alarm":("type":"ppu","action":"ХР"),"condition":("set":"TRUE","reset":"FALSE","active":"NOT dipar.U_AM.value"))'}
	N_U_AM : Talarm:= (subsystem_num := 10, type_num := 4); //Нет сигнала: Контроль питания ИМ//Нет DI/Блок управления
	{attribute 'export' := '("archive":"True","name":"Нет сигнала: Контроль питания аппаратуры вибрации, =24 В","alarm":("type":"ppu","action":"ХР"),"condition":("set":"TRUE","reset":"FALSE","active":"NOT dipar.Uvs_24.value"))'}
	N_Uvs_24 : Talarm:= (subsystem_num := 10, type_num := 4); //Нет сигнала: Контроль питания аппаратуры вибрации, =24 В//Нет DI/Блок управления
	{attribute 'export' := '("archive":"True","name":"Нет сигнала: Контроль питания дополнительного оборудования, =24В","alarm":("type":"ppu","action":"ХР"),"condition":("set":"TRUE","reset":"FALSE","active":"NOT dipar.Uother_24.value"))'}
	N_Uother_24 : Talarm:= (subsystem_num := 10, type_num := 4); //Нет сигнала: Контроль питания дополнительного оборудования, =24В//Нет DI/Блок управления
	{attribute 'export' := '("archive":"True","name":"Нет сигнала: Контроль питания ИМ2","alarm":("type":"ppu","action":"ХР"),"condition":("set":"TRUE","reset":"FALSE","active":"NOT dipar.U_AM2.value"))'}
	N_U_AM2 : Talarm:= (subsystem_num := 10, type_num := 4); //Нет сигнала: Контроль питания ИМ2//Нет DI/Блок управления
	{attribute 'export' := '("archive":"True","name":"Нет сигнала: Контроль питания ТРК рез.","alarm":("type":"ppu","action":"ХР"),"condition":("set":"TRUE","reset":"FALSE","active":"NOT dipar.Utrk_res.value"))'}
	N_Utrk_res : Talarm:= (subsystem_num := 10, type_num := 4); //Нет сигнала: Контроль питания ТРК рез.//Нет DI/Блок управления
	{attribute 'export' := '("archive":"True","name":"БЭО. Перегрузка фильтра EV3 (Осн. БЭО)","alarm":("type":"ppu","action":"ХР"),"condition":("set":"TRUE","reset":"FALSE","active":"dipar.EV3.value"))'}
	EV3 : Talarm:= (subsystem_num := 10, type_num := 4); //БЭО. Перегрузка фильтра EV3 (Осн. БЭО)//DI/Блок управления
	{attribute 'export' := '("archive":"True","name":"БЭО. Перегрузка фильтра EV4 (Рез. БЭО)","alarm":("type":"ppu","action":"ХР"),"condition":("set":"TRUE","reset":"FALSE","active":"dipar.EV4.value"))'}
	EV4 : Talarm:= (subsystem_num := 10, type_num := 4); //БЭО. Перегрузка фильтра EV4 (Рез. БЭО)//DI/Блок управления
	{attribute 'export' := '("archive":"True","name":"Нет сигнала: БЭО. Контроль основного ввода питания БЭО (-KV3)","alarm":("type":"ppu","action":"ХР"),"condition":("set":"TRUE","reset":"FALSE","active":"NOT dipar.Ubeo_main.value"))'}
	N_Ubeo_main : Talarm:= (subsystem_num := 10, type_num := 4); //Нет сигнала: БЭО. Контроль основного ввода питания БЭО (-KV3)//Нет DI/Блок управления
	{attribute 'export' := '("archive":"True","name":"Нет сигнала: БЭО. Контроль резервного ввода питания БЭО (-KV4)","alarm":("type":"ppu","action":"ХР"),"condition":("set":"TRUE","reset":"FALSE","active":"NOT dipar.Ubeo_res.value"))'}
	N_Ubeo_res : Talarm:= (subsystem_num := 10, type_num := 4); //Нет сигнала: БЭО. Контроль резервного ввода питания БЭО (-KV4)//Нет DI/Блок управления
	{attribute 'export' := '("archive":"True","name":"Нет сигнала: БЭО. Контроль -AG11","alarm":("type":"ppu","action":"ХР"),"condition":("set":"TRUE","reset":"FALSE","active":"NOT dipar.AG11.value"))'}
	N_AG11 : Talarm:= (subsystem_num := 10, type_num := 4); //Нет сигнала: БЭО. Контроль -AG11//Нет DI/Блок управления
	{attribute 'export' := '("archive":"True","name":"Нет сигнала: БЭО. Контроль -AG12","alarm":("type":"ppu","action":"ХР"),"condition":("set":"TRUE","reset":"FALSE","active":"NOT dipar.AG12.value"))'}
	N_AG12 : Talarm:= (subsystem_num := 10, type_num := 4); //Нет сигнала: БЭО. Контроль -AG12//Нет DI/Блок управления
	{attribute 'export' := '("archive":"True","name":"БЭО. Контроль замыкания на землю питания БЭО (-KR5)","alarm":("type":"ppu","action":"ХР"),"condition":("set":"TRUE","reset":"FALSE","active":"dipar.U_G_KR5.value"))'}
	U_G_KR5 : Talarm:= (subsystem_num := 10, type_num := 4); //БЭО. Контроль замыкания на землю питания БЭО (-KR5)//DI/Блок управления
	{attribute 'export' := '("archive":"True","name":"Нет сигнала: БЭО. Контроль питания кн. ЭАО","alarm":("type":"ppu","action":"ХР"),"condition":("set":"TRUE","reset":"FALSE","active":"NOT dipar.U_KEAO.value"))'}
	N_U_KEAO : Talarm:= (subsystem_num := 10, type_num := 4); //Нет сигнала: БЭО. Контроль питания кн. ЭАО//Нет DI/Блок управления
	{attribute 'export' := '("archive":"True","name":"Нет сигнала: БЭО. Контроль питания БЭО","alarm":("type":"ppu","action":"ХР"),"condition":("set":"TRUE","reset":"FALSE","active":"NOT dipar.U_BEO.value"))'}
	N_U_BEO : Talarm:= (subsystem_num := 10, type_num := 4); //Нет сигнала: БЭО. Контроль питания БЭО//Нет DI/Блок управления
	{attribute 'export' := '("archive":"True","name":"Нет сигнала: БЭО. Контроль питания БЗА","alarm":("type":"ppu","action":"ХР"),"condition":("set":"TRUE","reset":"FALSE","active":"NOT dipar.U_BZA.value"))'}
	N_U_BZA : Talarm:= (subsystem_num := 10, type_num := 4); //Нет сигнала: БЭО. Контроль питания БЗА//Нет DI/Блок управления
	{attribute 'export' := '("archive":"True","name":"Ошибка -AUO1","alarm":("type":"ppu","action":"ХР"),"condition":("set":"TRUE","reset":"FALSE","active":"dipar.Err_AUO1.value"))'}
	Err_AUO1 : Talarm:= (subsystem_num := 10, type_num := 4); //Ошибка -AUO1//DI/Блок управления
	{attribute 'export' := '("archive":"True","name":"Кран №1 не закрыт","alarm":("type":"ppu","action":"ХР"),"condition":("set":"TRUE","reset":"FALSE","active":"NOT dipar.Kr1_off.value OR dipar.Kr1_ON.value"))'}
	Kr1_off : Talarm:= (subsystem_num := 11, type_num := 4); //Кран №1 не закрыт//ALG/Газовая обвязка
	{attribute 'export' := '("archive":"True","name":"Кран №2 не закрыт","alarm":("type":"ppu","action":"ХР"),"condition":("set":"TRUE","reset":"FALSE","active":"NOT dipar.Kr2_off.value OR dipar.Kr2_ON.value"))'}
	Kr2_off : Talarm:= (subsystem_num := 11, type_num := 4); //Кран №2 не закрыт//ALG/Газовая обвязка
	{attribute 'export' := '("archive":"True","name":"Кран №4 не закрыт","alarm":("type":"ppu","action":"ХР"),"condition":("set":"TRUE","reset":"FALSE","active":"(NOT dipar.Kr4_off.value OR dipar.Kr4_ON.value) AND tch.nGas_N.value"))'}
	Kr4_off : Talarm:= (subsystem_num := 11, type_num := 4); //Кран №4 не закрыт//ALG/Газовая обвязка
	{attribute 'export' := '("archive":"True","name":"Кран №5 не открыт","alarm":("type":"ppu","action":"ХР"),"condition":("set":"TRUE","reset":"FALSE","active":"(NOT dipar.Kr5_ON.value OR dipar.Kr5_off.value) AND tch.nGas_N.value"))'}
	Kr5_ON : Talarm:= (subsystem_num := 11, type_num := 4); //Кран №5 не открыт//ALG/Газовая обвязка
	{attribute 'export' := '("archive":"True","name":"Кран №5 не закрыт","alarm":("type":"ppu","action":"ХР"),"condition":("set":"TRUE","reset":"FALSE","active":"(NOT dipar.Kr5_off.value OR dipar.Kr5_ON.value) AND tch.Gas_N.value"))'}
	Kr5_off : Talarm:= (subsystem_num := 11, type_num := 4); //Кран №5 не закрыт//ALG/Газовая обвязка
	{attribute 'export' := '("archive":"True","name":"Кран №6 не закрыт","alarm":("type":"ppu","action":"ХР"),"condition":("set":"TRUE","reset":"FALSE","active":"(NOT dipar.Kr6_off.value OR dipar.Kr6_ON.value) AND tch.nGas_N.value"))'}
	Kr6_off : Talarm:= (subsystem_num := 11, type_num := 4); //Кран №6 не закрыт//ALG/Газовая обвязка
END_VAR
(* global variable list trs *)
{region INFO}
(*
 Назначение: Признаки срабатывания аварийных сигнализаций, не приводящих к останову
 Автор:  /Andrey/ 24.06.2025 16:50:31
 Версия: v00.00.22
 Проект: KA107__GPA2
*)
{endregion}
{attribute 'qualified_only'}
{attribute 'symbol' := 'read'}
VAR_GLOBAL
	{attribute 'symbol' := 'none'}
	common : Talarm; //Общий сигнал для VAR_STAT

END_VAR
(* global variable list am *)
{region INFO}
(*
 Назначение:   Используется для хранения, инициализации и передачи на ВУ состояния исполнительных механизмов
 Автор:        /Разработчик/ 08.08.2025 8:32:24
 Конфигуратор: v00.01.00
 Проект:       KA107
*)
{endregion}
{attribute 'qualified_only'}
{attribute 'symbol' := 'readwrite'}
VAR_GLOBAL
	{attribute 'symbol' := 'none'}
	common : Tam;
	{attribute 'export' := '("name":"Вытяжной вентилятор ВОУ","tag":"","group":"Блок двигателя","actuator":("gender":"муж","action":"вкл/откл","prm":("name":["Всегда"],"alg":"true")))'}
	VV_VOU : TAM_2x1 := (subsystem_num := 2, PT_offOutTimeOn := t#1s, PT_offOutTimeOff := t#1s, PT_onDelay := t#0s, PT_offDelay := t#0s, PT_alertTimeOn := t#2s, PT_alertTimeOff := t#2s, onSig_inv := FALSE); //Вытяжной вентилятор ВОУ/2x1
	{attribute 'export' := '("name":"Вентилятор 1 АВОМ","tag":"","group":"Аппарат воздушного охлаждения масла двигателя","actuator":("gender":"муж","action":"вкл/откл","prm":("name":["Всегда"],"alg":"true")))'}
	Vn1_AVOM : TAM_2x1 := (subsystem_num := 5, PT_offOutTimeOn := t#1s, PT_offOutTimeOff := t#1s, PT_onDelay := t#0s, PT_offDelay := t#0s, PT_alertTimeOn := t#2s, PT_alertTimeOff := t#2s, onSig_inv := FALSE); //Вентилятор 1 АВОМ/2x1
	{attribute 'export' := '("name":"Вентилятор 2 АВОМ","tag":"","group":"Аппарат воздушного охлаждения масла двигателя","actuator":("gender":"муж","action":"вкл/откл","prm":("name":["Всегда"],"alg":"true")))'}
	Vn2_AVOM : TAM_2x1 := (subsystem_num := 5, PT_offOutTimeOn := t#1s, PT_offOutTimeOff := t#1s, PT_onDelay := t#0s, PT_offDelay := t#0s, PT_alertTimeOn := t#2s, PT_alertTimeOff := t#2s, onSig_inv := FALSE); //Вентилятор 2 АВОМ/2x1
	{attribute 'export' := '("name":"Вентилятор 3 АВОМ","tag":"","group":"Аппарат воздушного охлаждения масла двигателя","actuator":("gender":"муж","action":"вкл/откл","prm":("name":["Всегда"],"alg":"true")))'}
	Vn3_AVOM : TAM_2x1 := (subsystem_num := 5, PT_offOutTimeOn := t#1s, PT_offOutTimeOff := t#1s, PT_onDelay := t#0s, PT_offDelay := t#0s, PT_alertTimeOn := t#2s, PT_alertTimeOff := t#2s, onSig_inv := FALSE); //Вентилятор 3 АВОМ/2x1
	{attribute 'export' := '("name":"Вентилятор 4 АВОМ","tag":"","group":"Аппарат воздушного охлаждения масла двигателя","actuator":("gender":"муж","action":"вкл/откл","prm":("name":["Всегда"],"alg":"true")))'}
	Vn4_AVOM : TAM_2x1 := (subsystem_num := 5, PT_offOutTimeOn := t#1s, PT_offOutTimeOff := t#1s, PT_onDelay := t#0s, PT_offDelay := t#0s, PT_alertTimeOn := t#2s, PT_alertTimeOff := t#2s, onSig_inv := FALSE); //Вентилятор 4 АВОМ/2x1
	{attribute 'export' := '("communication":("unsubscribe":"OpTime"),"name":"Кран 1","tag":"","group":"Газовая обвязка","actuator":("gender":"муж","action":"откр/закр","prm":("name":[" Нет активных режимов"],"alg":"alg.V_000")))'}
	Kr1 : TAM_2x2 := (subsystem_num := 11, PT_offOutTimeOn := t#6s, PT_offOutTimeOff := t#6s, PT_onDelay := t#5s, PT_offDelay := t#5s, PT_alertTimeOn := t#11s, PT_alertTimeOff := t#11s); //Кран 1/2x2
	{attribute 'export' := '("communication":("unsubscribe":"OpTime"),"name":"Кран 2","tag":"","group":"Газовая обвязка","actuator":("gender":"муж","action":"откр/закр","prm":("name":[" Нет активных режимов"],"alg":"alg.V_000")))'}
	Kr2 : TAM_2x2 := (subsystem_num := 11, PT_offOutTimeOn := t#50s, PT_offOutTimeOff := t#50s, PT_onDelay := t#2s, PT_offDelay := t#2s, PT_alertTimeOn := t#60s, PT_alertTimeOff := t#60s); //Кран 2/2x2
	{attribute 'export' := '("communication":("unsubscribe":"OpTime"),"name":"Кран 4","tag":"","group":"Газовая обвязка","actuator":("gender":"муж","action":"откр/закр","prm":("name":[" Нет активных режимов"],"alg":"alg.V_000")))'}
	Kr4 : TAM_2x2 := (subsystem_num := 11, PT_offOutTimeOn := t#5s, PT_offOutTimeOff := t#5s, PT_onDelay := t#5s, PT_offDelay := t#5s, PT_alertTimeOn := t#10s, PT_alertTimeOff := t#10s); //Кран 4/2x2
	{attribute 'export' := '("communication":("unsubscribe":"OpTime"),"name":"Кран 5","tag":"","group":"Газовая обвязка","actuator":("gender":"муж","action":"откр/закр","prm":("name":[" Нет активных режимов"],"alg":"alg.V_000")))'}
	Kr5 : TAM_2x2 := (subsystem_num := 11, PT_offOutTimeOn := t#5s, PT_offOutTimeOff := t#5s, PT_onDelay := t#5s, PT_offDelay := t#5s, PT_alertTimeOn := t#10s, PT_alertTimeOff := t#10s); //Кран 5/2x2
	{attribute 'export' := '("communication":("unsubscribe":"OpTime"),"name":"Кран 6","tag":"","group":"Газовая обвязка","actuator":("gender":"муж","action":"откр/закр","prm":("name":[" Нет активных режимов"],"alg":"alg.V_000 OR mde.M AND NOT dipar.Kr6_Off.value AND dipar.Kr2_ON.value")))'}
	Kr6 : TAM_2x2 := (subsystem_num := 11, PT_offOutTimeOn := t#5s, PT_offOutTimeOff := t#5s, PT_onDelay := t#5s, PT_offDelay := t#5s, PT_alertTimeOn := t#10s, PT_alertTimeOff := t#10s); //Кран 6/2x2
	{attribute 'export' := '("communication":("unsubscribe":"OpTime"),"name":"Кран 12","tag":"","group":"Газовая обвязка","actuator":("gender":"муж","action":"откр/закр","prm":("name":[" Нет активных режимов"],"alg":"alg.V_000")))'}
	Kr12 : TAM_2x2 := (subsystem_num := 11, PT_offOutTimeOn := t#5s, PT_offOutTimeOff := t#5s, PT_onDelay := t#5s, PT_offDelay := t#5s, PT_alertTimeOn := t#10s, PT_alertTimeOff := t#10s); //Кран 12/2x2
	{attribute 'export' := '("communication":("unsubscribe":"OpTime"),"name":"Кран 9","tag":"","group":"Газовая обвязка","actuator":("gender":"муж","action":"откр/закр","prm":("name":["Никогда"],"alg":"FALSE")))'}
	Kr9 : TAM_2x2 := (subsystem_num := 11, PT_offOutTimeOn := t#5s, PT_offOutTimeOff := t#5s, PT_onDelay := t#5s, PT_offDelay := t#5s, PT_alertTimeOn := t#10s, PT_alertTimeOff := t#10s); //Кран 9/2x2
	{attribute 'export' := '("communication":("unsubscribe":"OpTime"),"name":"Кран 11","tag":"","group":"Газовая обвязка","actuator":("gender":"муж","action":"откр/закр","prm":("name":[" Нет активных режимов"],"alg":"alg.V_000")))'}
	Kr11 : TAM_2x2 := (subsystem_num := 11, PT_offOutTimeOn := t#5s, PT_offOutTimeOff := t#5s, PT_onDelay := t#5s, PT_offDelay := t#5s, PT_alertTimeOn := t#10s, PT_alertTimeOff := t#10s); //Кран 11/2x2
	{attribute 'export' := '("communication":("unsubscribe":"OpTime"),"name":"Кран 10","tag":"","group":"Газовая обвязка","actuator":("gender":"муж","action":"откр/закр","prm":("name":["Никогда"],"alg":"FALSE")))'}
	Kr10 : TAM_2x2 := (subsystem_num := 11, PT_offOutTimeOn := t#5s, PT_offOutTimeOff := t#5s, PT_onDelay := t#5s, PT_offDelay := t#5s, PT_alertTimeOn := t#10s, PT_alertTimeOff := t#10s); //Кран 10/2x2
	{attribute 'export' := '("communication":("unsubscribe":"OpTime"),"name":"КПВ 1","tag":"","group":"Блок двигателя","actuator":("gender":"муж","action":"откр/закр","reversed":"True","prm":("name":[" Нет активных режимов"],"alg":"alg.V_000")))'}
	KPV1 : TAM_1x2 := (subsystem_num := 2, PT_alertTimeOn := t#5s, PT_alertTimeOff := t#5s); //КПВ 1/1x2
	{attribute 'export' := '("communication":("unsubscribe":"OpTime"),"name":"КПВ 2","tag":"","group":"Блок двигателя","actuator":("gender":"муж","action":"откр/закр","reversed":"True","prm":("name":[" Нет активных режимов"],"alg":"alg.V_000")))'}
	KPV2 : TAM_1x2 := (subsystem_num := 2, PT_alertTimeOn := t#5s, PT_alertTimeOff := t#5s); //КПВ 2/1x2
	{attribute 'export' := '("communication":("unsubscribe":"OpTime"),"name":"КПВ 3","tag":"","group":"Блок двигателя","actuator":("gender":"муж","action":"откр/закр","reversed":"True","prm":("name":[" Нет активных режимов"],"alg":"alg.V_000")))'}
	KPV3 : TAM_1x2 := (subsystem_num := 2, PT_alertTimeOn := t#5s, PT_alertTimeOff := t#5s); //КПВ 3/1x2
	{attribute 'export' := '("communication":("unsubscribe":"OpTime"),"name":"КПВ 4","tag":"","group":"Блок двигателя","actuator":("gender":"муж","action":"откр/закр","reversed":"True","prm":("name":[" Нет активных режимов"],"alg":"alg.V_000")))'}
	KPV4 : TAM_1x2 := (subsystem_num := 2, PT_alertTimeOn := t#5s, PT_alertTimeOff := t#5s); //КПВ 4/1x2
	{attribute 'export' := '("communication":("unsubscribe":"OpTime"),"name":"КПВ 5","tag":"","group":"Блок двигателя","actuator":("gender":"муж","action":"откр/закр","reversed":"True","prm":("name":[" Нет активных режимов"],"alg":"alg.V_000")))'}
	KPV5 : TAM_1x2 := (subsystem_num := 2, PT_alertTimeOn := t#5s, PT_alertTimeOff := t#5s); //КПВ 5/1x2
	{attribute 'export' := '("communication":("unsubscribe":"OpTime"),"name":"Стопорный клапан","tag":"","group":"Блок топливного газа","actuator":("gender":"муж","action":"откр/закр","prm":("name":[" Нет активных режимов"],"alg":"alg.V_000")))'}
	SK : TAM_1x2 := (subsystem_num := 6, PT_alertTimeOn := t#2s, PT_alertTimeOff := t#2s); //Стопорный клапан/1x2
	{attribute 'export' := '("name":"Пусковой насос смазки","tag":"","group":"Маслосистема двигателя","actuator":("gender":"муж","action":"вкл/откл","prm":("name":["Всегда"],"alg":"true")))'}
	PNS : TAM_2x1 := (subsystem_num := 3, PT_offOutTimeOn := t#1s, PT_offOutTimeOff := t#1s, PT_onDelay := t#0s, PT_offDelay := t#0s, PT_alertTimeOn := t#2s, PT_alertTimeOff := t#2s, onSig_inv := FALSE); //Пусковой насос смазки/2x1
	{attribute 'export' := '("name":"Пусковой насос уплотнения","tag":"","group":"Компрессорная установка/блок нагнетателя","actuator":("gender":"муж","action":"вкл/откл","prm":("name":["Всегда"],"alg":"true")))'}
	PNU : TAM_2x1 := (subsystem_num := 9, PT_offOutTimeOn := t#1s, PT_offOutTimeOff := t#1s, PT_onDelay := t#0s, PT_offDelay := t#0s, PT_alertTimeOn := t#2s, PT_alertTimeOff := t#2s, onSig_inv := FALSE); //Пусковой насос уплотнения/2x1
	{attribute 'export' := '("communication":("unsubscribe":"OpTime"),"name":"ВНА","tag":"","group":"Блок двигателя","actuator":("gender":"муж","action":"откр/закр","prm":("name":[" Нет активных режимов"],"alg":"alg.V_000")))'}
	VNA : TAM_1x0 := (subsystem_num := 2); //ВНА/1x0
	{attribute 'export' := '("communication":("unsubscribe":"OpTime"),"name":"Звуковая сигнализация","tag":"","group":"Блок управления","actuator":("gender":"жен","action":"вкл/откл","prm":("name":[" Нет активных режимов"],"alg":"alg.V_000")))'}
	Sound : TAM_1x0 := (subsystem_num := 10); //Звуковая сигнализация/1x0
	{attribute 'export' := '("communication":("unsubscribe":"OpTime"),"name":"Агрегат зажигания","tag":"","group":"Блок двигателя","actuator":("gender":"муж","action":"вкл/откл","prm":("name":[" Нет активных режимов"],"alg":"alg.V_000")))'}
	AZ : TAM_1x0 := (subsystem_num := 2); //Агрегат зажигания/1x0
	{attribute 'export' := '("communication":("unsubscribe":"OpTime"),"name":"Обогрев ВНА","tag":"","group":"Блок двигателя","actuator":("gender":"муж","action":"вкл/откл","prm":("name":[" Нет активных режимов"],"alg":"alg.V_000")))'}
	VNA_heat : TAM_1x0 := (subsystem_num := 2); //Обогрев ВНА/1x0
	{attribute 'export' := '("communication":("unsubscribe":"OpTime"),"name":"Кран 13","tag":"","group":"Газовая обвязка","actuator":("gender":"муж","action":"откр/закр","prm":("name":[" Нет активных режимов"],"alg":"alg.V_000")))'}
	Kr13 : TAM_1x1 := (subsystem_num := 11, PT_alertTimeOn := t#3s, PT_alertTimeOff := t#3s, onSig_inv := FALSE); //Кран 13/1x1
	{attribute 'export' := '("communication":("unsubscribe":"OpTime"),"name":"Кран 15","tag":"","group":"Газовая обвязка","actuator":("gender":"муж","action":"откр/закр","prm":("name":[" Нет активных режимов"],"alg":"alg.V_000")))'}
	Kr15 : TAM_1x0 := (subsystem_num := 11); //Кран 15/1x0
	{attribute 'export' := '("name":"Вытяжной вентилятор нагнетателя","tag":"","group":"Компрессорная установка/блок нагнетателя","actuator":("gender":"муж","action":"вкл/откл","prm":("name":["Всегда"],"alg":"true")))'}
	VVN : TAM_2x1 := (subsystem_num := 9, PT_offOutTimeOn := t#1s, PT_offOutTimeOff := t#1s, PT_onDelay := t#0s, PT_offDelay := t#0s, PT_alertTimeOn := t#2s, PT_alertTimeOff := t#2s, onSig_inv := FALSE); //Вытяжной вентилятор нагнетателя/2x1
	{attribute 'export' := '("communication":("unsubscribe":"OpTime"),"name":"Дозатор газа","tag":"","group":"Блок двигателя","actuator":("prm":("name":["Нет активных режимов"],"alg":"alg.V_000")))'}
	DG : TAM_a := (subsystem_num := 2, isAcmd := TRUE, isReverse := FALSE); //Дозатор газа/a
END_VAR
(* global variable list acpar *)
{region INFO}
(*
 Назначение:    Используется для хранения, инициализации и передачи на ВУ состояния расчетных аналоговых параметров
 Автор:        /Разработчик/ 08.08.2025 8:32:24
 Конфигуратор: v00.01.00
 Проект:       KA107
*)
{endregion}
{attribute 'qualified_only'}
{attribute 'symbol' := 'readwrite'}
VAR_GLOBAL
	{attribute 'export' := '("archive":"True","communication":("cycle":"base"),"name":("full":"Расчётная Nтк","short":"Nтк"),"unit":"об/мин","tag":"","digit":"0","group":"Блок двигателя")'}
	Ntk : Tacpar := (setpoint := (activation_flags := 32, HHV := 8400, HHV_default := 8400), cfg := (lolim := 0, hilim := 9375)); //Расчётная Nтк//HHV := 8400/Блок двигателя
	{attribute 'export' := '("archive":"True","communication":("cycle":"base"),"name":("full":"Расчётная Nст","short":"Nст"),"unit":"об/мин","tag":"","digit":"0","group":"Блок двигателя")'}
	Nst : Tacpar := (setpoint := (activation_flags := 40, HV := 8500, HV_default := 8500, HHV := 9300, HHV_default := 9300), cfg := (lolim := 0, hilim := 9375)); //Расчётная Nст//HV := 8500, HHV := 9300/Блок двигателя
	{attribute 'export' := '("archive":"True","communication":("cycle":"base"),"name":("full":"Расчётная Тг перед СТ","short":"Тг"),"unit":"°C","tag":"","digit":"0","group":"Блок двигателя")'}
	Tg_inST : Tacpar := (setpoint := (activation_flags := 40, HV := 570, HV_default := 570, HHV := 670, HHV_default := 670), cfg := (lolim := -50, hilim := 1000)); //Расчётная Тг перед СТ//HV := 570, HHV := 670/Блок двигателя
	{attribute 'export' := '("archive":"True","communication":("cycle":"base"),"name":("full":"Приведенная Nгг","short":"Nгг"),"unit":"об/мин","tag":"","digit":"0","group":"Блок двигателя")'}
	NtkPrived : Tacpar := (setpoint := (activation_flags := 0), cfg := (lolim := 0, hilim := 13000)); //Приведенная Nгг///Блок двигателя
	{attribute 'export' := '("archive":"True","communication":("cycle":"base"),"name":("full":"Расход топливного газа","short":"Qтг"),"unit":"м3/ч","tag":"","digit":"0","group":"Блок двигателя")'}
	Qtg_m3 : Tacpar := (setpoint := (activation_flags := 0), cfg := (lolim := 0, hilim := 10000)); //Расход топливного газа///Блок двигателя
END_VAR
(* global variable list tunpar *)
{region INFO}
(*
 Назначение:   Используется для хранения, инициализации состояния аналоговых параметров, передаваемых с ВУ
 Автор:        /Разработчик/ 08.08.2025 8:32:24
 Конфигуратор: v00.01.00
 Проект:       KA107
*)
{endregion}
{attribute 'qualified_only'}
{attribute 'symbol' := 'readwrite'}
VAR_GLOBAL
	{attribute 'export' := '("archive":"True","communication":("cycle":"base"),"name":"Задание Nst","unit":"об/мин","digit":"0","limit":("low":"0","high":"8500"),"group":"Блок двигателя")'}
	setNst : Ttunpar := (value := 0, set_value := 0, enable_valueLimit := TRUE, lolim := 0, hilim := 8500); //Задание Nst/Блок двигателя
	{attribute 'export' := '("archive":"True","communication":("cycle":"base"),"name":"Задание Ntk","unit":"об/мин","digit":"0","limit":("low":"0","high":"8400"),"group":"Блок двигателя")'}
	setNtk : Ttunpar := (value := 0, set_value := 0, enable_valueLimit := TRUE, lolim := 0, hilim := 8400); //Задание Ntk/Блок двигателя
	{attribute 'export' := '("archive":"True","communication":("cycle":"base"),"name":"Шаг Nst для РЧВ","unit":"об/мин","digit":"0","limit":("low":"5","high":"50"),"group":"Блок двигателя")'}
	rateNstBtn : Ttunpar := (value := 30, set_value := 30, enable_valueLimit := TRUE, lolim := 5, hilim := 50); //Шаг Nst для РЧВ/Блок двигателя
	{attribute 'export' := '("archive":"True","communication":("cycle":"base"),"name":"Шаг Ntk для РЧВ","unit":"об/мин","digit":"0","limit":("low":"5","high":"30"),"group":"Блок двигателя")'}
	rateNtkBtn : Ttunpar := (value := 20, set_value := 20, enable_valueLimit := TRUE, lolim := 5, hilim := 30); //Шаг Ntk для РЧВ/Блок двигателя
	{attribute 'export' := '("archive":"True","communication":("cycle":"base"),"name":"Задание температуры маслосистемы","unit":"С","digit":"0","limit":("low":"20","high":"45"),"group":"Блок двигателя")'}
	setTm : Ttunpar := (value := 35, set_value := 35, enable_valueLimit := TRUE, lolim := 20, hilim := 45); //Задание температуры маслосистемы/Блок двигателя
	{attribute 'export' := '("archive":"True","communication":("cycle":"base"),"name":"Т1 ПИД АВОМ","unit":"","digit":"2","limit":("low":"0.01","high":"1"),"group":"АВОМ")'}
	T1_avom : Ttunpar := (value := 0.1, set_value := 0.1, enable_valueLimit := TRUE, lolim := 0.01, hilim := 1); //Т1 ПИД АВОМ/АВОМ
	{attribute 'export' := '("archive":"True","communication":("cycle":"base"),"name":"Т2 ПИД АВОМ","unit":"","digit":"0","limit":("low":"0.01","high":"1000"),"group":"АВОМ")'}
	T2_avom : Ttunpar := (value := 400, set_value := 400, enable_valueLimit := TRUE, lolim := 0.01, hilim := 1000); //Т2 ПИД АВОМ/АВОМ
	{attribute 'export' := '("archive":"True","communication":("cycle":"base"),"name":"К ПИД АВОМ","unit":"","digit":"2","limit":("low":"0.01","high":"1"),"group":"АВОМ")'}
	K_avom : Ttunpar := (value := 0.01, set_value := 0.01, enable_valueLimit := TRUE, lolim := 0.01, hilim := 1); //К ПИД АВОМ/АВОМ
	{attribute 'export' := '("archive":"True","communication":("cycle":"base"),"name":"Зона нечувствительности ПИД АВОМ","unit":"","digit":"1","limit":("low":"0.01","high":"10"),"group":"АВОМ")'}
	DZ_avom : Ttunpar := (value := 5, set_value := 5, enable_valueLimit := TRUE, lolim := 0.01, hilim := 10); //Зона нечувствительности ПИД АВОМ/АВОМ
	{attribute 'export' := '("archive":"True","communication":("cycle":"base"),"name":"Температура в маслобаке смазки","unit":"С","digit":"0","limit":("low":"5","high":"60"),"group":"Маслосистема Д")'}
	setTmMBDN : Ttunpar := (value := 50, set_value := 50, enable_valueLimit := TRUE, lolim := 5, hilim := 60); //Температура в маслобаке смазки/Маслосистема Д
	{attribute 'export' := '("archive":"True","communication":("cycle":"base"),"name":"Температура в маслобаке уплотнений","unit":"С","digit":"0","limit":("low":"5","high":"60"),"group":"Маслосистема К")'}
	setTmMBN : Ttunpar := (value := 50, set_value := 50, enable_valueLimit := TRUE, lolim := 5, hilim := 60); //Температура в маслобаке уплотнений/Маслосистема К
	{attribute 'export' := '("archive":"True","communication":("cycle":"slow"),"name":"Количество пусков","unit":"","digit":"0","limit":("low":"0","high":"1000000"),"group":"Наработки")'}
	countStart : Ttunpar := (value := 0, set_value := 0, enable_valueLimit := TRUE, lolim := 0, hilim := 1000000); //Количество пусков/Наработки
	{attribute 'export' := '("archive":"True","communication":("cycle":"slow"),"name":"Количество НО","unit":"","digit":"0","limit":("low":"0","high":"1000000"),"group":"Наработки")'}
	countNO : Ttunpar := (value := 0, set_value := 0, enable_valueLimit := TRUE, lolim := 0, hilim := 1000000); //Количество НО/Наработки
	{attribute 'export' := '("archive":"True","communication":("cycle":"slow"),"name":"Количество АО","unit":"","digit":"0","limit":("low":"0","high":"1000000"),"group":"Наработки")'}
	countAO : Ttunpar := (value := 0, set_value := 0, enable_valueLimit := TRUE, lolim := 0, hilim := 1000000); //Количество АО/Наработки
	{attribute 'export' := '("archive":"True","communication":("cycle":"slow"),"name":"Наработка суммарная","unit":"ч","digit":"0","limit":("low":"0","high":"1000000"),"group":"Наработки")'}
	generalOpTime : Ttunpar := (value := 0, set_value := 0, enable_valueLimit := TRUE, lolim := 0, hilim := 1000000); //Наработка суммарная/Наработки
	{attribute 'export' := '("archive":"True","communication":("cycle":"slow"),"name":"Наработка на режиме","unit":"ч","digit":"0","limit":("low":"0","high":"1000000"),"group":"Наработки")'}
	workOpTime : Ttunpar := (value := 0, set_value := 0, enable_valueLimit := TRUE, lolim := 0, hilim := 1000000); //Наработка на режиме/Наработки
END_VAR
(* global variable list btn *)
{region INFO}
(*
 Назначение:   Используется для хранения, инициализации и передачи на ВУ состояния кнопок
 Автор:        /Разработчик/ 08.08.2025 8:32:24
 Конфигуратор: v00.01.00
 Проект:       KA107
*)
{endregion}
{attribute 'qualified_only'}
{attribute 'symbol' := 'readwrite'}
VAR_GLOBAL
	{attribute 'export' := '("archive":"True","communication":("cycle":"base"),"name":"Имитацию включить","prm":("name":["Режим \"Ремонт\""],"alg":"mde.Repair"))'}
	imit_ON : Tbtn; //Имитацию включить
	{attribute 'export' := '("archive":"True","communication":("cycle":"base"),"name":"Имитацию выключить","prm":("name":["Логическая 1"],"alg":"TRUE"))'}
	imit_OF : Tbtn; //Имитацию выключить
	{attribute 'export' := '("archive":"True","communication":("cycle":"base"),"name":"Тестирование включить","prm":("name":["Режим \"Ремонт\""],"alg":"mde.Repair"))'}
	test_on : Tbtn; //Тестирование включить
	{attribute 'export' := '("archive":"True","communication":("cycle":"base"),"name":"Тестирование выключить","prm":("name":["Логическая 1"],"alg":"TRUE"))'}
	test_off : Tbtn; //Тестирование выключить
	{attribute 'export' := '("archive":"True","communication":("cycle":"base"),"name":"Ремонт","prm":("name":["Режим \"ХР\" ИЛИ Режим \"ГР\""],"alg":"alg.V_000 AND NOT tch.PrepareStart.value"))'}
	Repair : Tbtn; //Ремонт
	{attribute 'export' := '("archive":"True","communication":("cycle":"base"),"name":"Холодный резерв","prm":("name":["Режим \"Ремонт\" ИЛИ Режим \"ГР\""],"alg":"( mde.Repair OR mde.GR ) AND NOT tch.PrepareStart.value AND NOT tch.CheckAlarm_on.Value "))'}
	HR : Tbtn; //Холодный резерв
	{attribute 'export' := '("archive":"True","communication":("cycle":"base"),"name":"Горячий резерв","prm":("name":["Режим \"Ремонт\" ИЛИ Режим \"ХР\""],"alg":"mde.Repair OR mde.HR AND NOT tch.CheckAlarm_on.Value "))'}
	GR : Tbtn; //Горячий резерв
	{attribute 'export' := '("archive":"True","communication":("cycle":"base"),"name":"Комплексная проверка кранов","prm":("name":["Режим \"ГР\""],"alg":"mde.GR AND NOT ( tch.PrepareStart.value OR tch.Gas_N.value )"))'}
	KPK : Tbtn; //Комплексная проверка кранов
	{attribute 'export' := '("archive":"True","communication":("cycle":"base"),"name":"Холодная прокрутка","prm":("name":["Режим \"ХР\" ИЛИ Режим \"ГР\""],"alg":"mde.GR AND NOT tch.PrepareStart.value"))'}
	HP : Tbtn; //Холодная прокрутка
	{attribute 'export' := '("archive":"True","communication":("cycle":"base"),"name":"Автоматический пуск на Кольцо","prm":("name":["Режим \"ГР\""],"alg":"mde.GR AND NOT tch.PrepareStart.value"))'}
	APK : Tbtn; //Автоматический пуск на Кольцо
	{attribute 'export' := '("archive":"True","communication":("cycle":"base"),"name":"Пуск","prm":("name":["Выбран один из пусковых режимов и есть готовность к пуску после \"Контроля САУ\""],"alg":"check.ReadytoSF AND check.prm_start"))'}
	Start : Tbtn; //Пуск
	{attribute 'export' := '("archive":"True","communication":("cycle":"base"),"name":"Отмена","prm":("name":["Выбран один из пусковых режимов"],"alg":"check.ReadytoSF OR mde.Repair OR check.tmrCancelPrm.Q"))'}
	Cancel : Tbtn; //Отмена
	{attribute 'export' := '("archive":"True","communication":("cycle":"base"),"name":"Контроль САУ","prm":("name":["Логическая 1"],"alg":"TRUE"))'}
	Check_SAU : Tbtn; //Контроль САУ
	{attribute 'export' := '("archive":"True","communication":("cycle":"base"),"name":"Переход Магистраль-Кольцо","prm":("name":["Режим \"Магистраль\" ИЛИ Режим \"Переход К-М\""],"alg":"mde.M OR mde.K_M"))'}
	M_K : Tbtn; //Переход Магистраль-Кольцо
	{attribute 'export' := '("archive":"True","communication":("cycle":"base"),"name":"Переход Кольцо-Магистраль","prm":("name":["Режим \"Кольцо\" ИЛИ Режим \"Переход М-К\""],"alg":"mde.K OR mde.M_K"))'}
	K_M : Tbtn; //Переход Кольцо-Магистраль
	{attribute 'export' := '("archive":"True","communication":("cycle":"base"),"name":"Нормальный останов со стравливанием","prm":("name":["Рабочие режимы ИЛИ Режим \"НОбс\""],"alg":"alg.work OR mde.NObs"))'}
	NOss : Tbtn; //Нормальный останов со стравливанием
	{attribute 'export' := '("archive":"True","communication":("cycle":"base"),"name":"Нормальный останов без стравливания","prm":("name":["Рабочие режимы"],"alg":"alg.work"))'}
	NObs : Tbtn; //Нормальный останов без стравливания
	{attribute 'export' := '("archive":"True","communication":("cycle":"base"),"name":"Аварийный останов со стравливанием","prm":("name":["Логическая 1"],"alg":"TRUE"))'}
	AOss : Tbtn; //Аварийный останов со стравливанием
	{attribute 'export' := '("archive":"True","communication":("cycle":"base"),"name":"Аварийный останов без стравливания","prm":("name":["Нет Режима \"АОсс\""],"alg":"NOT mde.AOss"))'}
	AObs : Tbtn; //Аварийный останов без стравливания
	{attribute 'export' := '("archive":"True","communication":("cycle":"base"),"name":"Деблокировка","prm":("name":["Логическая 1"],"alg":"TRUE"))'}
	Unlock : Tbtn; //Деблокировка
	{attribute 'export' := '("archive":"True","communication":("cycle":"base"),"name":"РЧВ: вверх","prm":("name":["Режим ТР \"Работа\""],"alg":"tch.GTDwork.value"))'}
	turnUP : Tbtn; //РЧВ: вверх
	{attribute 'export' := '("archive":"True","communication":("cycle":"base"),"name":"РЧВ: вниз","prm":("name":["Режим ТР \"Работа\""],"alg":"tch.GTDwork.value"))'}
	turnDN : Tbtn; //РЧВ: вниз
	{attribute 'export' := '("archive":"True","communication":("cycle":"base"),"name":"Запись настроек регулятора","prm":("name":["Не нажата кнопка \"Считывание настроек\""],"alg":"NOT btn.get_tun.out"))'}
	set_tun : Tbtn; //Запись настроек регулятора
	{attribute 'export' := '("archive":"True","communication":("cycle":"base"),"name":"Считывание настроек регулятора","prm":("name":["Не нажата кнопка \"Запись настроек\""],"alg":"NOT btn.set_tun.out"))'}
	get_tun : Tbtn; //Считывание настроек регулятора
	{attribute 'export' := '("archive":"True","communication":("cycle":"base"),"name":"Стравливание","prm":("name":["Нет активных режимов"],"alg":"alg.V_000"))'}
	bleeding : Tbtn; //Стравливание
	{attribute 'export' := '("archive":"True","communication":("cycle":"base"),"name":"Проверку защит включить","prm":("name":["Режим \"Ремонт\""],"alg":"mde.Repair"))'}
	CheckAlarm_on : Tbtn; //Проверку защит включить
	{attribute 'export' := '("archive":"True","communication":("cycle":"base"),"name":"Проверку защит выключить","prm":("name":["Режим \"Ремонт\""],"alg":"mde.Repair"))'}
	CheckAlarm_off : Tbtn; //Проверку защит выключить
END_VAR
(* global variable list mde *)
{region INFO}
(*
 Назначение:   Используется для хранения и передачи на ВУ режимов
 Автор:        /Разработчик/ 08.08.2025 8:32:24
 Конфигуратор: v00.01.00
 Проект:       KA107
*)
{endregion}
{attribute 'qualified_only'}
{attribute 'symbol' := 'none'}
VAR_GLOBAL
	number : ENUM_MODE; //Текущий режим
	AOss : BOOL; //Аварийный останов со стравливанием газа
	AObs : BOOL; //Аварийный останов без стравливания газа
	NOss : BOOL; //Нормальный останов со стравливанием газа
	NObs : BOOL; //Нормальный останов без стравливания газа
	Repair : BOOL; //Техническое обслуживание и текущий ремонт
	HR : BOOL; //Холодный резерв
	GR : BOOL; //Горячий резерв
	PZ : BOOL; //Проверка защит
	HP : BOOL; //Холодная прокрутка
	KPK : BOOL; //Комплексная проверка кранов
	APK : BOOL; //Автоматический пуск на «Кольцо»
	K : BOOL; //Кольцо
	M : BOOL; //Магистраль
	K_M : BOOL; //Переход «Кольцо - Магистраль»
	M_K : BOOL; //Переход «Магистраль - Кольцо»
	Error : BOOL; //Нет режима (ошибка)
END_VAR
(* global variable list aipar *)
{region INFO}
(*
 Назначение: Используется для хранения, инициализации и передачи на ВУ значений и состояния входных аналоговых параметров
 Автор:      /Andrey/ 16.07.2025 17:15:05
 Версия ТЭ5: v00.00.01
 Проект:     KA107
*)
{endregion}
{attribute 'qualified_only'}
{attribute 'symbol' := 'readwrite'}
VAR_GLOBAL
	{attribute 'symbol' := 'none'}
	common : Taipar;
	{attribute 'export' := '("archive":"True","communication":("cycle":"fast","unsubscribe":["setpoint.LLV","setpoint.L1V","setpoint.LV","setpoint.HV","setpoint.H1V","setpoint.HHV"]),"journal":"True","name":("full":"Частота вращения ТК канал 1","short":"ЧВ ТК кан.1"),"unit":("engineering":"об/мин","electrical":"Гц"),"digit":"1","connection":("module":"UCP1-A1-FI1-1","type":"F","device_clamp":"UCP1","clamp":"XFI1:1А XFI1:1В XFI1:3А"),"subsystem":"Блок двигателя","group":["Блок двигателя"])'}
	Ntk_1 : Taipar := (setpoint := (activation_flags := 0), cfg := (par_type := 6, lolim := 0, hilim := 9375, k := 2.342)); //Частота вращения ТК канал 1///Уставки//
	{attribute 'export' := '("archive":"True","communication":("cycle":"fast","unsubscribe":["setpoint.LLV","setpoint.L1V","setpoint.LV","setpoint.HV","setpoint.H1V","setpoint.HHV"]),"journal":"True","name":("full":"Частота вращения СТ канал 1","short":"ЧВ СТ кан.1"),"unit":("engineering":"об/мин","electrical":"Гц"),"digit":"1","connection":("module":"UCP1-A1-FI1-2","type":"F","device_clamp":"UCP1","clamp":"XFI1:4A XFI1:4B XFI1:6A"),"subsystem":"Блок двигателя","group":["Блок двигателя"])'}
	Nst_1 : Taipar := (setpoint := (activation_flags := 0), cfg := (par_type := 6, lolim := 0, hilim := 9375, k := 2.342)); //Частота вращения СТ канал 1///Уставки//
	{attribute 'export' := '("archive":"True","communication":("cycle":"fast","unsubscribe":["setpoint.LLV","setpoint.L1V","setpoint.LV","setpoint.HV","setpoint.H1V","setpoint.HHV"]),"journal":"True","name":("full":"Частота вращения ТК канал 2","short":"ЧВ ТК кан.2"),"unit":("engineering":"об/мин","electrical":"Гц"),"digit":"1","connection":("module":"UCP1-A1-FI2-1","type":"F","device_clamp":"UCP1","clamp":"XFI1:10A XFI1:10B XFI1:12A"),"subsystem":"Блок двигателя","group":["Блок двигателя"])'}
	Ntk_2 : Taipar := (setpoint := (activation_flags := 0), cfg := (par_type := 6, lolim := 0, hilim := 9375, k := 2.342)); //Частота вращения ТК канал 2///Уставки//
	{attribute 'export' := '("archive":"True","communication":("cycle":"fast","unsubscribe":["setpoint.LLV","setpoint.L1V","setpoint.LV","setpoint.HV","setpoint.H1V","setpoint.HHV"]),"journal":"True","name":("full":"Частота вращения СТ канал 2","short":"ЧВ СТ кан.2"),"unit":("engineering":"об/мин","electrical":"Гц"),"digit":"1","connection":("module":"UCP1-A1-FI2-2","type":"F","device_clamp":"UCP1","clamp":"XFI1:13A XFI1:13B XFI1:15A"),"subsystem":"Блок двигателя","group":["Блок двигателя"])'}
	Nst_2 : Taipar := (setpoint := (activation_flags := 0), cfg := (par_type := 6, lolim := 0, hilim := 9375, k := 2.342)); //Частота вращения СТ канал 2///Уставки//
	{attribute 'export' := '("archive":"True","communication":("cycle":"fast","unsubscribe":["setpoint.LLV","setpoint.L1V","setpoint.LV","setpoint.H1V"]),"journal":"True","name":("full":"Виброскорость ТК","short":"Виброск. ТК"),"unit":("engineering":"мм/с","electrical":"мА"),"digit":"1","connection":("module":"UCP1-A1-AI1-1","type":"I, акт.","device_clamp":"UCP1","clamp":"XAI1:1A XAI1:1B"),"subsystem":"Блок двигателя","group":["Блок двигателя"])'}
	Vstk : Taipar := (setpoint := (activation_flags := 40, HV := 50, HV_default := 50, HHV := 60, HHV_default := 60, hyst := GVL_LIB.Hyst_SP), cfg := (par_type := 1, lolim := 0, hilim := 100)); //Виброскорость ТК///Уставки//HV := 50/HHV := 60/
	{attribute 'export' := '("archive":"True","communication":("cycle":"fast","unsubscribe":["setpoint.LLV","setpoint.L1V","setpoint.LV","setpoint.H1V"]),"journal":"True","name":("full":"Виброскорость СТ","short":"Виброск. СТ"),"unit":("engineering":"мм/с","electrical":"мА"),"digit":"1","connection":("module":"UCP1-A1-AI1-2","type":"I, акт.","device_clamp":"UCP1","clamp":"XAI1:2A XAI1:2B"),"subsystem":"Блок двигателя","group":["Блок двигателя"])'}
	Vsst : Taipar := (setpoint := (activation_flags := 40, HV := 50, HV_default := 50, HHV := 60, HHV_default := 60, hyst := GVL_LIB.Hyst_SP), cfg := (par_type := 1, lolim := 0, hilim := 100)); //Виброскорость СТ///Уставки//HV := 50/HHV := 60/
	{attribute 'export' := '("archive":"True","communication":("cycle":"fast","unsubscribe":["setpoint.LLV","setpoint.L1V","setpoint.LV","setpoint.HV","setpoint.H1V","setpoint.HHV"]),"journal":"True","name":("full":"Положение топливного клапана дозатора газа","short":"Пол. ДГ"),"unit":("engineering":"%","electrical":"мА"),"digit":"1","connection":("module":"UCP1-A1-AI1-3","type":"I, акт.","device_clamp":"UCP1","clamp":"XAI1:3A XAI1:3B"),"subsystem":"Блок двигателя","group":["Блок двигателя"])'}
	DG_pos : Taipar := (setpoint := (activation_flags := 0, hyst := GVL_LIB.Hyst_SP), cfg := (par_type := 1, lolim := 0, hilim := 100)); //Положение топливного клапана дозатора газа///Уставки//
	{attribute 'export' := '("archive":"True","communication":("cycle":"base","unsubscribe":["setpoint.L1V","setpoint.HV","setpoint.H1V","setpoint.HHV"]),"journal":"True","name":("full":"Перепад давления “масло-газ”","short":"dP масло-газ"),"unit":("engineering":"МПа","electrical":"мА"),"digit":"1","connection":("module":"UCP1-A1-AI1-4","type":"I, акт.","device_clamp":"UCP1","clamp":"Внутр. сигнал"),"subsystem":"Блок компрессора","group":["Блок компрессора"])'}
	dPmg : Taipar := (setpoint := (activation_flags := 5, LLV := 0.3, LLV_default := 0.3, LV := 0.5, LV_default := 0.5, hyst := GVL_LIB.Hyst_SP), cfg := (par_type := 1, lolim := 0, hilim := 4)); //Перепад давления “масло-газ”///Уставки//LLV := 0.3/LV := 0.5/
	{attribute 'export' := '("archive":"True","communication":("cycle":"fast","unsubscribe":["setpoint.LLV","setpoint.L1V","setpoint.LV","setpoint.HV","setpoint.H1V","setpoint.HHV"]),"journal":"True","name":("full":"диаг. (Сигнал управления положением дозатора газа)","short":"Пол. ДГ (диаг)"),"unit":("engineering":"%","electrical":"мА"),"digit":"1","connection":("module":"UCP1-A1-AI1-8","type":"I, акт.","device_clamp":"UCP1","clamp":"Внутр. сигнал"),"subsystem":"Блок автоматики","group":["Блок автоматики"])'}
	DG_pos_diag : Taipar := (setpoint := (activation_flags := 0), cfg := (par_type := 1, lolim := 0, hilim := 100)); //диаг. (Сигнал управления положением дозатора газа)///Уставки//
	{attribute 'export' := '("archive":"True","communication":("cycle":"fast","unsubscribe":["setpoint.LLV","setpoint.L1V","setpoint.LV","setpoint.HV","setpoint.H1V"]),"journal":"True","name":("full":"Давление воздуха за 14-й ступенью осевого компрессора","short":"Давл. за компр."),"unit":("engineering":"МПа","electrical":"мА"),"digit":"1","connection":("module":"UCP1-A1-AI2-1","type":"I, пас.","device_clamp":"UCP1","clamp":"XAI3:1A XAI3:1B"),"subsystem":"Блок двигателя","group":["Блок двигателя"])'}
	Pa_out14 : Taipar := (setpoint := (activation_flags := 32, HHV := 1.99, HHV_default := 1.99, hyst := GVL_LIB.Hyst_SP), cfg := (par_type := 1, lolim := 0, hilim := 2)); //Давление воздуха за 14-й ступенью осевого компрессора///Уставки//HHV := 1.99/
	{attribute 'export' := '("archive":"True","communication":("cycle":"base","unsubscribe":["setpoint.LLV","setpoint.L1V","setpoint.LV","setpoint.HV","setpoint.H1V","setpoint.HHV"]),"journal":"True","name":("full":"Давление газа на входе Н","short":"Pg на входе Н"),"unit":("engineering":"МПа","electrical":"мА"),"digit":"1","connection":("module":"UCP1-A1-AI2-2","type":"I, акт.","device_clamp":"UCP1","clamp":"Внутр. сигнал"),"subsystem":"Газовая обвязка","group":["Газовая обвязка"])'}
	Pg_inN : Taipar := (setpoint := (activation_flags := 0, hyst := GVL_LIB.Hyst_SP), cfg := (par_type := 1, lolim := 0, hilim := 6)); //Давление газа на входе Н///Уставки//
	{attribute 'export' := '("archive":"True","communication":("cycle":"base","unsubscribe":["setpoint.LLV","setpoint.L1V","setpoint.LV","setpoint.HV","setpoint.H1V","setpoint.HHV"]),"journal":"True","name":("full":"Давление газа на выходе Н","short":"Pg на выходе Н"),"unit":("engineering":"МПа","electrical":"мА"),"digit":"1","connection":("module":"UCP1-A1-AI2-3","type":"I, акт.","device_clamp":"UCP1","clamp":"Внутр. сигнал"),"subsystem":"Газовая обвязка","group":["Газовая обвязка"])'}
	Pg_outN : Taipar := (setpoint := (activation_flags := 0, hyst := GVL_LIB.Hyst_SP), cfg := (par_type := 1, lolim := 0, hilim := 10)); //Давление газа на выходе Н///Уставки//
	{attribute 'export' := '("archive":"True","communication":("cycle":"base","unsubscribe":["setpoint.LLV","setpoint.L1V","setpoint.LV","setpoint.HV","setpoint.H1V","setpoint.HHV"]),"journal":"True","name":("full":"Температура газа на входе Н","short":"Pg на входе Н"),"unit":("engineering":"°С","electrical":"мА"),"digit":"1","connection":("module":"UCP1-A1-AI2-4","type":"I, акт.","device_clamp":"UCP1","clamp":"Внутр. сигнал"),"subsystem":"Газовая обвязка","group":["Газовая обвязка"])'}
	Tg_inN : Taipar := (setpoint := (activation_flags := 0, hyst := GVL_LIB.Hyst_SP), cfg := (par_type := 1, lolim := -50, hilim := 50)); //Температура газа на входе Н///Уставки//
	{attribute 'export' := '("archive":"True","communication":("cycle":"base","unsubscribe":["setpoint.LLV","setpoint.L1V","setpoint.LV","setpoint.HV","setpoint.H1V","setpoint.HHV"]),"journal":"True","name":("full":"Температура газа на выходе Н","short":"Pg на выходе Н"),"unit":("engineering":"°С","electrical":"мА"),"digit":"1","connection":("module":"UCP1-A1-AI2-5","type":"I, акт.","device_clamp":"UCP1","clamp":"Внутр. сигнал"),"subsystem":"Газовая обвязка","group":["Газовая обвязка"])'}
	Tg_outN : Taipar := (setpoint := (activation_flags := 0, hyst := GVL_LIB.Hyst_SP), cfg := (par_type := 1, lolim := -50, hilim := 100)); //Температура газа на выходе Н///Уставки//
	{attribute 'export' := '("archive":"True","communication":("cycle":"fast","unsubscribe":["setpoint.LLV","setpoint.L1V","setpoint.LV","setpoint.HV","setpoint.H1V","setpoint.HHV"]),"journal":"True","name":("full":"Перепад давления на конфузоре","short":"dP конфузоп"),"unit":("engineering":"кПа","electrical":"мА"),"digit":"1","connection":("module":"UCP1-A1-AI2-6","type":"I, акт.","device_clamp":"UCP1","clamp":"Внутр. сигнал"),"subsystem":"Газовая обвязка","group":["Газовая обвязка"])'}
	dP_conf : Taipar := (setpoint := (activation_flags := 0, hyst := GVL_LIB.Hyst_SP), cfg := (par_type := 1, lolim := 0, hilim := 60)); //Перепад давления на конфузоре///Уставки//
	{attribute 'export' := '("archive":"True","communication":("cycle":"base","unsubscribe":["setpoint.LLV","setpoint.L1V","setpoint.LV","setpoint.HV","setpoint.H1V","setpoint.HHV"]),"journal":"True","name":("full":"Влажность атмосферного воздуха в блоке автоматики","short":"H воздуха"),"unit":("engineering":"%","electrical":"мА"),"tag":"ПВТ100","digit":"1","connection":("module":"UCP1-A1-AI3-2","type":"I, акт.","device_clamp":"UCP1","clamp":"Внутр. сигнал"),"subsystem":"Блок автоматики","group":["Блок автоматики"])'}
	Vlaz_BA : Taipar := (setpoint := (activation_flags := 0, hyst := GVL_LIB.Hyst_SP), cfg := (par_type := 1, lolim := 0, hilim := 100)); //Влажность атмосферного воздуха в блоке автоматики/ПВТ100//Уставки//
	{attribute 'export' := '("archive":"True","communication":("cycle":"base","unsubscribe":["setpoint.LLV","setpoint.L1V","setpoint.LV","setpoint.HV","setpoint.H1V","setpoint.HHV"]),"journal":"True","name":("full":"Температура атмосферного воздуха в блоке автоматики, нижняя часть","short":"t воздуха"),"unit":("engineering":"°С","electrical":"мА"),"tag":"ПВТ100","digit":"1","connection":("module":"UCP1-A1-AI3-3","type":"I, акт.","device_clamp":"UCP1","clamp":"Внутр. сигнал"),"subsystem":"Блок автоматики","group":["Блок автоматики"])'}
	Ta_BAdown : Taipar := (setpoint := (activation_flags := 0, hyst := GVL_LIB.Hyst_SP), cfg := (par_type := 1, lolim := 0, hilim := 100)); //Температура атмосферного воздуха в блоке автоматики, нижняя часть/ПВТ100//Уставки//
	{attribute 'export' := '("archive":"True","communication":("cycle":"base","unsubscribe":["setpoint.LLV","setpoint.L1V","setpoint.LV","setpoint.HV","setpoint.H1V","setpoint.HHV"]),"journal":"True","name":("full":"Температура атмосферного воздуха в блоке автоматики, верхняя часть","short":"t воздуха"),"unit":("engineering":"°С","electrical":"мА"),"tag":"ПВТ100","digit":"1","connection":("module":"UCP1-A1-AI3-4","type":"I, акт.","device_clamp":"UCP1","clamp":"Внутр. сигнал"),"subsystem":"Блок автоматики","group":["Блок автоматики"])'}
	Ta_BAup : Taipar := (setpoint := (activation_flags := 0, hyst := GVL_LIB.Hyst_SP), cfg := (par_type := 1, lolim := 0, hilim := 100)); //Температура атмосферного воздуха в блоке автоматики, верхняя часть/ПВТ100//Уставки//
	{attribute 'export' := '("archive":"True","communication":("cycle":"base","unsubscribe":["setpoint.L1V","setpoint.H1V","setpoint.HHV"]),"journal":"True","name":("full":"Давление топливного газа перед ТРК","short":"Ptg перед ДГ"),"unit":("engineering":"МПа","electrical":"мА"),"digit":"1","connection":("module":"UCP1-A1-AI3-5","type":"I, пас.","device_clamp":"UCP1","clamp":"FVP1:1 FVP1:2"),"subsystem":"Блок топливного газа","group":["Блок топливного газа"])'}
	Ptg_inTRK : Taipar := (setpoint := (activation_flags := 13, LLV := 1, LLV_default := 1, LV := 2, LV_default := 2, HV := 2.74, HV_default := 2.74, hyst := GVL_LIB.Hyst_SP), cfg := (par_type := 1, lolim := 0, hilim := 6)); //Давление топливного газа перед ТРК///Уставки//LLV := 1/LV := 2/HV := 2.74/
	{attribute 'export' := '("archive":"True","communication":("cycle":"base","unsubscribe":["setpoint.LLV","setpoint.L1V","setpoint.LV","setpoint.HV","setpoint.H1V","setpoint.HHV"]),"journal":"True","name":("full":"Перепад давления топливного газа на мерной шайбе ТГ","short":"dPtg"),"unit":("engineering":"кПа","electrical":"мА"),"digit":"1","connection":("module":"UCP1-A1-AI3-6","type":"I, пас.","device_clamp":"UCP1","clamp":"FVP1:3 FVP1:4"),"subsystem":"Блок топливного газа","group":["Блок топливного газа"])'}
	dPtg_inMD : Taipar := (setpoint := (activation_flags := 0, hyst := GVL_LIB.Hyst_SP), cfg := (par_type := 1, lolim := 0, hilim := 100)); //Перепад давления топливного газа на мерной шайбе ТГ///Уставки//
	{attribute 'export' := '("archive":"True","communication":("cycle":"base","unsubscribe":["setpoint.LLV","setpoint.L1V","setpoint.LV","setpoint.HV","setpoint.H1V","setpoint.HHV"]),"journal":"True","name":("full":"Температура холодного спая","short":"t хол. Спая"),"unit":("engineering":"°С","electrical":"°С"),"digit":"1","connection":("module":"UCP1-A1-AI4-1","type":"R","device_clamp":"UCP1","clamp":"Внутр. сигнал"),"subsystem":"Блок автоматики","group":["Блок автоматики"])'}
	Tcool : Taipar := (setpoint := (activation_flags := 0, hyst := GVL_LIB.Hyst_SP), cfg := (par_type := 4, lolim := -50, hilim := 200)); //Температура холодного спая///Уставки//
	{attribute 'export' := '("archive":"True","communication":("cycle":"base","unsubscribe":["setpoint.LLV","setpoint.L1V","setpoint.LV","setpoint.H1V","setpoint.HHV"]),"journal":"True","name":("full":"Температура упорного подшипника Н","short":"t упН"),"unit":("engineering":"°С","electrical":"°С"),"digit":"1","connection":("module":"UCP1-A1-AI4-2","type":"R","device_clamp":"UCP1","clamp":"FVT1:1 FVT1:3 FVT1:2"),"subsystem":"Блок компрессора","group":["Блок компрессора"])'}
	Tup_N : Taipar := (setpoint := (activation_flags := 8, HV := 80, HV_default := 80, hyst := GVL_LIB.Hyst_SP), cfg := (par_type := 4, lolim := -50, hilim := 500)); //Температура упорного подшипника Н///Уставки//HV := 80/
	{attribute 'export' := '("archive":"True","communication":("cycle":"base","unsubscribe":["setpoint.LLV","setpoint.L1V","setpoint.HV","setpoint.H1V","setpoint.HHV"]),"journal":"True","name":("full":"Температура масла на входе двигателя","short":"tm на вх. Д"),"unit":("engineering":"°С","electrical":"°С"),"digit":"1","connection":("module":"UCP1-A1-AI4-3","type":"R","device_clamp":"UCP1","clamp":"FVT2:1 FVT2:3 FVT2:2"),"subsystem":"Маслосистема Д","group":["Маслосистема Д"])'}
	Tm_inD : Taipar := (setpoint := (activation_flags := 4, LV := 40, LV_default := 40, hyst := GVL_LIB.Hyst_SP), cfg := (par_type := 4, lolim := -50, hilim := 500)); //Температура масла на входе двигателя///Уставки//LV := 40/
	{attribute 'export' := '("archive":"True","communication":("cycle":"base","unsubscribe":["setpoint.LLV","setpoint.L1V","setpoint.LV","setpoint.HV","setpoint.H1V"]),"journal":"True","name":("full":"Температура масла на выходе двигателя","short":"tm на вых. Д"),"unit":("engineering":"°С","electrical":"°С"),"digit":"1","connection":("module":"UCP1-A1-AI4-4","type":"R","device_clamp":"UCP1","clamp":"FVT3:1 FVT3:3 FVT3:2"),"subsystem":"Маслосистема Д","group":["Маслосистема Д"])'}
	Tm_outD : Taipar := (setpoint := (activation_flags := 32, HHV := 85, HHV_default := 85, hyst := GVL_LIB.Hyst_SP), cfg := (par_type := 4, lolim := -50, hilim := 500)); //Температура масла на выходе двигателя///Уставки//HHV := 85/
	{attribute 'export' := '("archive":"True","communication":("cycle":"base","unsubscribe":["setpoint.LLV","setpoint.L1V","setpoint.HV","setpoint.H1V","setpoint.HHV"]),"journal":"True","name":("full":"Температура масла в баке Д и Н","short":"tm в баке"),"unit":("engineering":"°С","electrical":"°С"),"digit":"1","connection":("module":"UCP1-A1-AI4-6","type":"R","device_clamp":"UCP1","clamp":"FVT5:1 FVT5:3 FVT5:2"),"subsystem":"Маслосистема Д","group":["Маслосистема Д"])'}
	Tm_MB : Taipar := (setpoint := (activation_flags := 4, LV := 5, LV_default := 5, hyst := GVL_LIB.Hyst_SP), cfg := (par_type := 4, lolim := -50, hilim := 500)); //Температура масла в баке Д и Н///Уставки//LV := 5/
	{attribute 'export' := '("archive":"True","communication":("cycle":"base","unsubscribe":["setpoint.LLV","setpoint.L1V","setpoint.HV","setpoint.H1V","setpoint.HHV"]),"journal":"True","name":("full":"Температура масла в баке уплотнения","short":"tm в баке"),"unit":("engineering":"°С","electrical":"°С"),"digit":"1","connection":("module":"UCP1-A1-AI4-7","type":"R","device_clamp":"UCP1","clamp":"FVT6:1 FVT6:3 FVT6:2"),"subsystem":"Маслосистема Д","group":["Маслосистема Д"])'}
	Tm_MBU : Taipar := (setpoint := (activation_flags := 4, LV := 5, LV_default := 5, hyst := GVL_LIB.Hyst_SP), cfg := (par_type := 4, lolim := -50, hilim := 500)); //Температура масла в баке уплотнения///Уставки//LV := 5/
	{attribute 'export' := '("archive":"True","communication":("cycle":"base","unsubscribe":["setpoint.LLV","setpoint.L1V","setpoint.LV","setpoint.H1V","setpoint.HHV"]),"journal":"True","name":("full":"Температура масла на выходе АВОМ Д и Н","short":"tm АВОМ"),"unit":("engineering":"°С","electrical":"°С"),"digit":"1","connection":("module":"UCP1-A1-AI4-8","type":"R","device_clamp":"UCP1","clamp":"FVT7:1 FVT7:3 FVT7:2"),"subsystem":"Маслосистема Д","group":["Маслосистема Д"])'}
	Tm_outAVOM : Taipar := (setpoint := (activation_flags := 8, HV := 80, HV_default := 80, hyst := GVL_LIB.Hyst_SP), cfg := (par_type := 4, lolim := -50, hilim := 500)); //Температура масла на выходе АВОМ Д и Н///Уставки//HV := 80/
	{attribute 'export' := '("archive":"True","communication":("cycle":"base","unsubscribe":["setpoint.LLV","setpoint.L1V","setpoint.LV","setpoint.HV","setpoint.H1V","setpoint.HHV"]),"journal":"True","name":("full":"Температура топливного газа","short":"t топ. Газа"),"unit":("engineering":"°С","electrical":"°С"),"digit":"1","connection":("module":"UCP1-A1-AI5-2","type":"R","device_clamp":"UCP1","clamp":"FVT9:1 FVT9:3 FVT9:2"),"subsystem":"Блок топливного газа","group":["Блок топливного газа"])'}
	Ttg : Taipar := (setpoint := (activation_flags := 0, hyst := GVL_LIB.Hyst_SP), cfg := (par_type := 4, lolim := -100, hilim := 200)); //Температура топливного газа///Уставки//
	{attribute 'export' := '("archive":"True","communication":("cycle":"base","unsubscribe":["setpoint.LLV","setpoint.L1V","setpoint.LV","setpoint.HV","setpoint.H1V","setpoint.HHV"]),"journal":"True","name":("full":"Температура масла на выходе АВОМ уплотнений","short":"tm АВОМ"),"unit":("engineering":"°С","electrical":"°С"),"digit":"1","connection":("module":"UCP1-A1-AI5-3","type":"R","device_clamp":"UCP1","clamp":"FVT10:1 FVT10:3 FVT10:2"),"subsystem":"Маслосистема К","group":["Маслосистема К"])'}
	Tm_outAU : Taipar := (setpoint := (activation_flags := 0, hyst := GVL_LIB.Hyst_SP), cfg := (par_type := 4, lolim := -50, hilim := 500)); //Температура масла на выходе АВОМ уплотнений///Уставки//
	{attribute 'export' := '("archive":"True","communication":("cycle":"base","unsubscribe":["setpoint.LLV","setpoint.L1V","setpoint.LV","setpoint.H1V","setpoint.HHV"]),"journal":"True","name":("full":"Температура опорного подшипника №1 Н","short":"t опН"),"unit":("engineering":"°С","electrical":"°С"),"digit":"1","connection":("module":"UCP1-A1-AI5-5","type":"R","device_clamp":"UCP1","clamp":"FVT12:1 FVT12:3 FVT12:2"),"subsystem":"Блок компрессора","group":["Блок компрессора"])'}
	Top_N_1 : Taipar := (setpoint := (activation_flags := 8, HV := 80, HV_default := 80, hyst := GVL_LIB.Hyst_SP), cfg := (par_type := 4, lolim := -50, hilim := 500)); //Температура опорного подшипника №1 Н///Уставки//HV := 80/
	{attribute 'export' := '("archive":"True","communication":("cycle":"base","unsubscribe":["setpoint.LLV","setpoint.L1V","setpoint.LV","setpoint.H1V","setpoint.HHV"]),"journal":"True","name":("full":"Температура опорного подшипника №2 Н","short":"t опН"),"unit":("engineering":"°С","electrical":"°С"),"digit":"1","connection":("module":"UCP1-A1-AI5-6","type":"R","device_clamp":"UCP1","clamp":"FVT13:1 FVT13:3 FVT13:2"),"subsystem":"Блок компрессора","group":["Блок компрессора"])'}
	Top_N_2 : Taipar := (setpoint := (activation_flags := 8, HV := 80, HV_default := 80, hyst := GVL_LIB.Hyst_SP), cfg := (par_type := 4, lolim := -50, hilim := 500)); //Температура опорного подшипника №2 Н///Уставки//HV := 80/
	{attribute 'export' := '("archive":"True","communication":("cycle":"base","unsubscribe":["setpoint.LLV","setpoint.L1V","setpoint.LV","setpoint.HV","setpoint.H1V","setpoint.HHV"]),"journal":"True","name":("full":"Температура газа на входе СТ 1 канал","short":"t на вх. СТ 1"),"unit":("engineering":"°С","electrical":"°С"),"digit":"1","connection":("module":"UCP1-A1-AI6-1","type":"TC","device_clamp":"UCP1","clamp":"XAI5:1A XAI5:1B"),"subsystem":"Блок двигателя","group":["Блок двигателя"])'}
	Tg_inST_1 : Taipar := (setpoint := (activation_flags := 0, hyst := GVL_LIB.Hyst_SP), cfg := (par_type := 5, lolim := -50, hilim := 1000, ucv_enabled := TRUE, ucvV := 10000)); //Температура газа на входе СТ 1 канал///Уставки//
	{attribute 'export' := '("archive":"True","communication":("cycle":"base","unsubscribe":["setpoint.LLV","setpoint.L1V","setpoint.LV","setpoint.HV","setpoint.H1V","setpoint.HHV"]),"journal":"True","name":("full":"Температура газа на входе СТ 3 канал","short":"t на вх. СТ 3"),"unit":("engineering":"°С","electrical":"°С"),"digit":"1","connection":("module":"UCP1-A1-AI6-2","type":"TC","device_clamp":"UCP1","clamp":"XAI5:2A XAI5:2B"),"subsystem":"Блок двигателя","group":["Блок двигателя"])'}
	Tg_inST_3 : Taipar := (setpoint := (activation_flags := 0, hyst := GVL_LIB.Hyst_SP), cfg := (par_type := 5, lolim := -50, hilim := 1000, ucv_enabled := TRUE, ucvV := 10000)); //Температура газа на входе СТ 3 канал///Уставки//
	{attribute 'export' := '("archive":"True","communication":("cycle":"base","unsubscribe":["setpoint.LLV","setpoint.L1V","setpoint.LV","setpoint.HV","setpoint.H1V","setpoint.HHV"]),"journal":"True","name":("full":"Температура газа на входе СТ 5 канал","short":"t на вх. СТ 5"),"unit":("engineering":"°С","electrical":"°С"),"digit":"1","connection":("module":"UCP1-A1-AI6-3","type":"TC","device_clamp":"UCP1","clamp":"XAI5:3A XAI5:3B"),"subsystem":"Блок двигателя","group":["Блок двигателя"])'}
	Tg_inST_5 : Taipar := (setpoint := (activation_flags := 0, hyst := GVL_LIB.Hyst_SP), cfg := (par_type := 5, lolim := -50, hilim := 1000, ucv_enabled := TRUE, ucvV := 10000)); //Температура газа на входе СТ 5 канал///Уставки//
	{attribute 'export' := '("archive":"True","communication":("cycle":"base","unsubscribe":["setpoint.LLV","setpoint.L1V","setpoint.LV","setpoint.HV","setpoint.H1V","setpoint.HHV"]),"journal":"True","name":("full":"Температура перед СК","short":"t перед СК"),"unit":("engineering":"°С","electrical":"°С"),"digit":"1","connection":("module":"UCP1-A1-AI6-5","type":"R","device_clamp":"UCP1","clamp":"XAI6:1A XAI6:1B XAI6:2B"),"subsystem":"Блок топливного газа","group":["Блок топливного газа"])'}
	Tg_inSK : Taipar := (setpoint := (activation_flags := 0, hyst := GVL_LIB.Hyst_SP), cfg := (par_type := 4, lolim := -100, hilim := 200)); //Температура перед СК///Уставки//
	{attribute 'export' := '("archive":"True","communication":("cycle":"base","unsubscribe":["setpoint.LLV","setpoint.L1V","setpoint.LV","setpoint.HV","setpoint.H1V","setpoint.HHV"]),"journal":"True","name":("full":"Температура газа на входе СТ 2 канал","short":"t на вх. СТ 2"),"unit":("engineering":"°С","electrical":"°С"),"digit":"1","connection":("module":"UCP1-A1-AI7-1","type":"TC","device_clamp":"UCP1","clamp":"XAI5:5A XAI5:5B"),"subsystem":"Блок двигателя","group":["Блок двигателя"])'}
	Tg_inST_2 : Taipar := (setpoint := (activation_flags := 0, hyst := GVL_LIB.Hyst_SP), cfg := (par_type := 5, lolim := -50, hilim := 1000, ucv_enabled := TRUE, ucvV := 10000)); //Температура газа на входе СТ 2 канал///Уставки//
	{attribute 'export' := '("archive":"True","communication":("cycle":"base","unsubscribe":["setpoint.LLV","setpoint.L1V","setpoint.LV","setpoint.HV","setpoint.H1V","setpoint.HHV"]),"journal":"True","name":("full":"Температура газа на входе СТ 4 канал","short":"t на вх. СТ 4"),"unit":("engineering":"°С","electrical":"°С"),"digit":"1","connection":("module":"UCP1-A1-AI7-2","type":"TC","device_clamp":"UCP1","clamp":"XAI5:6A XAI5:6B"),"subsystem":"Блок двигателя","group":["Блок двигателя"])'}
	Tg_inST_4 : Taipar := (setpoint := (activation_flags := 0, hyst := GVL_LIB.Hyst_SP), cfg := (par_type := 5, lolim := -50, hilim := 1000, ucv_enabled := TRUE, ucvV := 10000)); //Температура газа на входе СТ 4 канал///Уставки//
	{attribute 'export' := '("archive":"True","communication":("cycle":"base","unsubscribe":["setpoint.LLV","setpoint.L1V","setpoint.LV","setpoint.HV","setpoint.H1V","setpoint.HHV"]),"journal":"True","name":("full":"Температура газа на входе СТ 6 канал","short":"t на вх. СТ 6"),"unit":("engineering":"°С","electrical":"°С"),"digit":"1","connection":("module":"UCP1-A1-AI7-3","type":"TC","device_clamp":"UCP1","clamp":"XAI5:7A XAI5:7B"),"subsystem":"Блок двигателя","group":["Блок двигателя"])'}
	Tg_inST_6 : Taipar := (setpoint := (activation_flags := 0, hyst := GVL_LIB.Hyst_SP), cfg := (par_type := 5, lolim := -50, hilim := 1000, ucv_enabled := TRUE, ucvV := 10000)); //Температура газа на входе СТ 6 канал///Уставки//
